// ----------------------------------------------------
// Calculate maximum expected current
// ----------------------------------------------------
IF in_lrHeaterResistance > 0.0 THEN
    stat.lrMaxCurrent := SQRT(in_lrHeaterMaxPower / in_lrHeaterResistance);
ELSE
    stat.lrMaxCurrent := 999.9;
END_IF;


// ----------------------------------------------------
// Calculate expected heater power and power ratio
// ----------------------------------------------------
lrExpectedPower :=
    (stat.lrActSetpoint / 100.0) * in_lrHeaterMaxPower;

stat.lrExpectedHeaterPower := lrExpectedPower;

IF lrExpectedPower > 0.0 THEN
    lrPowerRatio := stat.lrActHeaterPower / lrExpectedPower;
ELSE
    lrPowerRatio := 1.0;
END_IF;

stat.lrHeaterPowerRatio := lrPowerRatio;


// ----------------------------------------------------
// Heater open-loop detection
// ----------------------------------------------------
// Below 1% demand, current measurement is not reliable enough.
stat.bHeaterOpenLoop :=
    (lrPowerRatio < 0.10)
    AND stat.bActive
    AND stat.lrActSetpoint > 1.0;


// ----------------------------------------------------
// Heater short-circuit detection
// ----------------------------------------------------
stat.bHeaterShort :=
    stat.lrActCurrent > (stat.lrMaxCurrent + 1.0);


// ----------------------------------------------------
// Thermal switch open detection
// ----------------------------------------------------
// One or more parallel heater branches may be disconnected.
// Actual power is reduced, but not zero.
bThermalSwitchOpenCandidate :=
    (lrPowerRatio >= 0.10)
    AND (lrPowerRatio < 0.85)
    AND stat.bActive
    AND stat.lrActSetpoint > 10.0
    AND NOT stat.bHeaterOpenLoop
    AND NOT stat.bHeaterShort;

// Debounce to avoid false alarms during transients
tonThermalSwitchOpen(
    IN := bThermalSwitchOpenCandidate,
    PT := T#10s
);

stat.bHeaterThermalSwitchOpen := tonThermalSwitchOpen.Q;


// ----------------------------------------------------
// Insufficient heater power
// ----------------------------------------------------
// Heater demand is high, but delivered power is too low.
// This means the heater may not be able to reach/hold setpoint.
stat.bHeaterInsufficientPower :=
    stat.bActive
    AND stat.lrActSetpoint > 50.0
    AND (lrPowerRatio < 0.70)
    AND NOT stat.bHeaterOpenLoop
    AND NOT stat.bHeaterShort;


// ----------------------------------------------------
// General error / warning flags
// ----------------------------------------------------
stat.bError :=
    stat.bHwError
    OR stat.bHeaterOpenLoop
    OR stat.bHeaterShort
    OR stat.bHeaterThermalSwitchOpen
    OR stat.bHeaterInsufficientPower;

stat.bWarning := stat.bHwWarning;


// ----------------------------------------------------
// Store auto setpoint information
// ----------------------------------------------------
stat.lrAutoSetpointValue := in_lrAutoSetpointValue;
stat.sAutoSetpointSource := in_sAutoSetpointSource;


// ----------------------------------------------------
// Set heater state
// ----------------------------------------------------
IF stat.bHwError THEN
    stat.nHeaterState := E_METIS_CRYO_HEATER_STATE.ERROR;
    stat.sHeaterState := 'HW ERROR';

ELSIF stat.bHeaterShort THEN
    stat.nHeaterState := E_METIS_CRYO_HEATER_STATE.ERROR;
    stat.sHeaterState := 'HEATER SHORT CIRCUIT';

ELSIF stat.bHeaterOpenLoop THEN
    stat.nHeaterState := E_METIS_CRYO_HEATER_STATE.ERROR;
    stat.sHeaterState := 'HEATER OPEN CIRCUIT';

ELSIF stat.bHeaterThermalSwitchOpen THEN
    stat.nHeaterState := E_METIS_CRYO_HEATER_STATE.ERROR;
    stat.sHeaterState := 'THERMAL SWITCH OPEN';

ELSIF stat.bHeaterInsufficientPower THEN
    stat.nHeaterState := E_METIS_CRYO_HEATER_STATE.ERROR;
    stat.sHeaterState := 'INSUFFICIENT HEATER POWER';

ELSIF stat.bHwWarning THEN
    stat.nHeaterState := E_METIS_CRYO_HEATER_STATE.ERROR;
    stat.sHeaterState := 'HW WARNING';

ELSIF stat.bWarning THEN
    stat.nHeaterState := E_METIS_CRYO_HEATER_STATE.ERROR;
    stat.sHeaterState := 'WARNING';

ELSIF stat.bManual THEN
    stat.nHeaterState := E_METIS_CRYO_HEATER_STATE.ON;
    stat.sHeaterState := 'MANUAL';

ELSIF stat.bActive THEN
    stat.nHeaterState := E_METIS_CRYO_HEATER_STATE.ON;
    stat.sHeaterState := 'ON';

ELSE
    stat.nHeaterState := E_METIS_CRYO_HEATER_STATE.OFF;
    stat.sHeaterState := 'OFF';
END_IF;


M_SetStatus := NOT stat.bError;


// stat.lrAutoCtrlOut := in_lrAutoSetpointValue;
// 
// 
// CASE in_eHeaterType OF
//     
//     E_METIS_CRYO_HEATER_TYPE.PWM_DETECTOR,
//     E_METIS_CRYO_HEATER_TYPE.PWM_WINDOW:
//         // Set actual power I * 24.0V
//         stat.lrActHeaterPower := stat.lrActCurrent * stat.lrActCurrent * in_lrHeaterResistance;
// 
//     E_METIS_CRYO_HEATER_TYPE.PWM_SORPTION:
//     
//         // Set actual power I^(Average PWM Voltage)
//         // TODO : CHECK IF CORRECT
//         stat.lrActHeaterPower := ((stat.lrActCurrent * 24 * stat.lrActDutyCycle)/100);
// 
//     E_METIS_CRYO_HEATER_TYPE.CPAU60:
//         // Set actual power I^2R
//         stat.lrActHeaterPower := stat.lrActCurrent * stat.lrActCurrent * in_lrHeaterResistance;
//         
//     E_METIS_CRYO_HEATER_TYPE.CXWUI60:
//         // Set actual power I^2R
//         stat.lrActHeaterPower := stat.lrActCurrent * stat.lrActCurrent * in_lrHeaterResistance;
// 
//     E_METIS_CRYO_HEATER_TYPE.EL95X1:
//         IF stat.bActive THEN
//             stat.lrActHeaterPower := stat.lrActCurrent * stat.lrActVoltage;
//         ELSE
//             stat.lrActHeaterPower := 0.0;
//         END_IF
//         
// END_CASE
// 
// // Set max current
// IF in_lrHeaterResistance > 0.0 THEN
//     stat.lrMaxCurrent :=  SQRT(in_lrHeaterMaxPower/in_lrHeaterResistance);
// ELSE
//     stat.lrMaxCurrent := 999.9;
// END_IF
// 
// // check if the heater is in open loop
// // Note: below 1.00% the current measurement is not accurate, so don't report an open loop error!
// stat.bHeaterOpenLoop := (stat.lrActHeaterPower < 0.1 * (stat.lrActSetpoint/100.0) * in_lrHeaterMaxPower) // actual power in [W] is less than 10% of the expected power in [W]
//                         AND stat.bActive 
//                         AND stat.lrActSetpoint > 1.0; // lrActSetpoint is more than 1% 
// 
// // Check if there is a short circuit: Comparing the actual current with the Max current + 1 A  
// stat.bHeaterShort := stat.lrActCurrent > (stat.lrMaxCurrent + 1);
// 
// // calculate the general bError/bWarning flags
// stat.bError := stat.bHwError OR stat.bHeaterOpenLoop OR stat.bHeaterShort;
// stat.bWarning := stat.bHwWarning;
// 
// stat.lrAutoSetpointValue := in_lrAutoSetpointValue;
// stat.sAutoSetpointSource := in_sAutoSetpointSource;
// 
// IF stat.bHwError THEN
//     stat.nHeaterState := E_METIS_CRYO_HEATER_STATE.ERROR;
//     stat.sHeaterState := 'HW ERROR';
// ELSIF stat.bHwWarning THEN
//     stat.nHeaterState := E_METIS_CRYO_HEATER_STATE.ERROR;
//     stat.sHeaterState := 'HW WARNING';
// ELSIF stat.bHeaterOpenLoop THEN
//     stat.nHeaterState := E_METIS_CRYO_HEATER_STATE.ERROR;
//     stat.sHeaterState := 'HEATER OPEN LOOP ERROR';
// ELSIF stat.bHeaterShort THEN
//     stat.nHeaterState := E_METIS_CRYO_HEATER_STATE.ERROR;
//     stat.sHeaterState := 'HEATER SHORT ERROR';
// ELSIF stat.bError THEN
//     stat.nHeaterState := E_METIS_CRYO_HEATER_STATE.ERROR;
//     stat.sHeaterState := 'ERROR';
// ELSIF stat.bWarning THEN
//     stat.nHeaterState := E_METIS_CRYO_HEATER_STATE.ERROR;
//     stat.sHeaterState := 'WARNING';
// ELSIF stat.bActive THEN
//     stat.nHeaterState := E_METIS_CRYO_HEATER_STATE.ON;
//     stat.sHeaterState := 'ON';
// ELSE
//     stat.nHeaterState := E_METIS_CRYO_HEATER_STATE.OFF;
//     stat.sHeaterState := 'OFF';
// END_IF
// 
//
END_METHOD

METHOD M_UpdateAlarms
VAR_INPUT
END_VAR
VAR
	stEventEntry : TcEventEntry;
	sText : STRING;
END_VAR
//
// Set / clear alarms
//

fbAlarmHandler.M_UpdateAlarm(
    in_bCondition    := stat.bHeaterShort,
    in_nIndex        := 0,
    in_strEventEntry := Tc_Events.METISCryoHeaterEventClass.HeaterShortCircuit
);

fbAlarmHandler.M_UpdateAlarm(
    in_bCondition    := stat.bHeaterOpenLoop,
    in_nIndex        := 1,
    in_strEventEntry := Tc_Events.METISCryoHeaterEventClass.HeaterOpenCircuit
);

fbAlarmHandler.M_UpdateAlarm(
    in_bCondition    := stat.bManual,
    in_nIndex        := 2,
    in_strEventEntry := Tc_Events.METISCryoHeaterEventClass.HeaterManualMode
);

fbAlarmHandler.M_UpdateAlarm(
    in_bCondition    := stat.bHeaterThermalSwitchOpen,
    in_nIndex        := 3,
    in_strEventEntry := Tc_Events.METISCryoHeaterEventClass.HeaterThermalSwitchOpen
);

fbAlarmHandler.M_UpdateAlarm(
    in_bCondition    := stat.bHeaterInsufficientPower,
    in_nIndex        := 4,
    in_strEventEntry := Tc_Events.METISCryoHeaterEventClass.HeaterInsufficientPower
);


//
// Handle alarms
//
fbAlarmHandler(stAlarms := stat.stAlarms);

fbAlarmHandler.M_ProcessAlarms(
    arrEventEntry := arrEventEntry,
    sEventString  := in_sName
);

// //
// // Set / clear alarms
// //
// 
// // Global alarm if the voted temperature reading is not valid.
// fbAlarmHandler.M_UpdateAlarm(
//     in_bCondition    := stat.bHeaterOpenLoop,
//     in_nIndex        := 1,
//     in_strEventEntry := Tc_Events.METISCryoHeaterEventClass.HeaterOpenCircuit
// );
// 
// 
// fbAlarmHandler.M_UpdateAlarm(
//     in_bCondition    := stat.bHeaterShort,
//     in_nIndex        := 0,
//     in_strEventEntry := Tc_Events.METISCryoHeaterEventClass.HeaterShortCircuit
// );
// 
// fbAlarmHandler.M_UpdateAlarm(
//     in_bCondition    := stat.bManual,
//     in_nIndex        := 2,
//     in_strEventEntry := Tc_Events.METISCryoHeaterEventClass.HeaterManualMode
// );
// 
// fbAlarmHandler.M_UpdateAlarm(
//     in_bCondition    := stat.,
//     in_nIndex        := 3,
//     in_strEventEntry := Tc_Events.METISCryoHeaterEventClass.HeaterThermalSwitchOpen
// );
// 
// fbAlarmHandler.M_UpdateAlarm(
//     in_bCondition    := stat.,
//     in_nIndex        := 4,
//     in_strEventEntry := Tc_Events.METISCryoHeaterEventClass.HeaterInsufficientPower
// );
// 
// 
// 
// 
// 
// //
// // Handle alarms
// //
// fbAlarmHandler(stAlarms := stat.stAlarms);
// 
// fbAlarmHandler.M_ProcessAlarms(
//     arrEventEntry := arrEventEntry,
//     sEventString  := in_sName
// );
END_METHOD

END_FUNCTION_BLOCK

// POUs/XML_Cfg_Read_Write/FB_READ_WRITE_HEATER_CONFIG
FUNCTION_BLOCK FB_READ_WRITE_HEATER_CONFIG EXTENDS FB_READ_WRITE_CONFIG_BASE
VAR_INPUT
	in_sHeaterName:      T_MaxString;
END_VAR
VAR_IN_OUT
	cfg:   T_METIS_HEATER_CFG;
END_VAR

SUPER^(
    in_sEntryName  := in_sHeaterName,
    in_sSubFolder  := 'Heater\',
    in_sXPath      := '/Heater_Configuration/',
    in_pSymAddr    := ADR(cfg),
    in_cbSymSize   := SIZEOF(cfg));

END_FUNCTION_BLOCK

// POUs/Devices/Control_Valves_Ctrl/FB_METIS_CONTROL_VALVE
FUNCTION_BLOCK FB_METIS_CONTROL_VALVE
VAR_INPUT
    {attribute 'OPC.UA.DA' := '0'}    
    in_sName:               STRING  := 'Ctrl Valve'; // Valve name
//    {attribute 'OPC.UA.DA' := '0'}
//    in_lrHeaterResistance:  LREAL;               // Resistance of the heater to be controlled [Ohms]
//    {attribute 'OPC.UA.DA' := '0'}
//    in_lrHeaterMaxPower:    LREAL;               // Max power of the heater to be controlled [Watts]    
    {attribute 'OPC.UA.DA' := '0'}

    in_eValveType:         		E_METIS_CRYO_CTRL_VALVE_TYPE := E_METIS_CRYO_Ctrl_VALVE_TYPE.NONE;
    {attribute 'OPC.UA.DA' := '0'}

    in_sAutoSetpointSource:     STRING;          // Name of the source of the AUTO setpoint
    
    {attribute 'OPC.UA.DA' := '0'}
    in_bEnable : BOOL;                           // Auto-mode enable
    
   {attribute 'OPC.UA.DA' := '0'}
   in_lrAutoSetpointValue:     LREAL;           // Output power coming for the AUTO setpoint
END_VAR
VAR
(*TODO: This input is useful if a PID ctrl loop is implemeted to control the valve.
For the moment, There are three set points, Off, Normal and Alarm*)	
// 	{attribute 'OPC.UA.DA' := '0'}
//     in_lrAutoSetpointValue:     LREAL;           // Output power coming for the AUTO setpoint
    {attribute 'OPC.UA.DA' := '0'}
    nTimeout:                   UDINT := 10000;     // Timeout for current to change [ms] after enabling power. Default 10000.
    {attribute 'OPC.UA.DA' := '0'}
	{attribute 'TcHmiSymbol.Show'}
    bInterlock:                 BOOL := FALSE;      // External Interlock
    {attribute 'OPC.UA.DA' := '0'}
    i_nCouplerState     AT %I*: UINT;               // Terminal state. Should be 8, i.e. OP.
// Hardware link    
    {attribute 'OPC.UA.DA' := '0'}
    io_anti_fog_blower      : T_METIS_CTRL_VALVE_IO_ANTI_FOG_BLOWER;
    {attribute 'OPC.UA.DA' := '0'}
    io_img_cfo_precooling   : T_METIS_CTRL_VALVE_IO_IMG_CFO_PRECOOLING;
    // EL2819 diagnostics for the output channel

    i_bOverTemperature  AT %I*: BOOL;
    i_bOpenLoad         AT %I*: BOOL;
    i_bOverCurrent      AT %I*: BOOL;
    i_bShortTo24V       AT %I*: BOOL;
	
//    {attribute 'OPC.UA.DA' := '0'}
//    io_cxwui60  : T_METIS_HEATER_IO_CXWUI60;
    
    {attribute 'OPC.UA.DA' := '1'}
	{attribute 'TcHmiSymbol.Show'}
    stat:        T_METIS_CTRL_VALVE_STAT;
    {attribute 'OPC.UA.DA' := '1'}
	{attribute 'TcHmiSymbol.ShowRecursively'}
    ctrl:        T_METIS_CTRL_VALVE_CTRL;
    {attribute 'OPC.UA.DA' := '1'}
	{attribute 'TcHmiSymbol.Show'}
		{attribute 'TcHmiSymbol.ShowRecursively'}
    cfg:         T_METIS_CTRL_VALVE_CFG;

    {attribute 'OPC.UA.DA' := '0'}
	{attribute 'TcHmiSymbol.Show'}
    fbConfig    : FB_READ_WRITE_CONTROL_VALVE_CONFIG; 
	
				// Alarm handling
	// List of alarms to be handled by Temperature
	arrEventEntry : ARRAY [0..3] OF TcEventEntry;
	// Alarm handler FB
	fbAlarmHandler : FB_AlarmHandler;
	{attribute 'TcHmiSymbol.Show'}
	{attribute 'TcHmiSymbol.ReadOnly'}
	sInstanceName : T_MaxString;
	{attribute 'TcHmiSymbol.Show'}
	bConfirmAllAlarms : BOOL;
	{attribute 'TcHmiSymbol.Show'}
	{attribute 'TcHmiSymbol.ReadOnly'}
	sEventClassName : T_MaxString;
	
	// Logs logs
	logs:	FB_CRYO_FUNCTION_LOG;
    
END_VAR

IF not stat.bConfigured THEN
    M_Configure();
END_IF

// Read/write the configuration
fbConfig(in_sCtrlValveName:= in_sName, cfg := cfg);

M_SetMode();

M_UpdateActive();

M_ReadInputs();

M_SetStatus();

M_SetCtrlOutput();

// read/write the config (if needed)
M_Read_Write_Config();

// Handle alarms
M_UpdateAlarms();

METHOD M_Activity_Valve_Alarm : BOOL
VAR_INPUT
END_VAR
in_lrAutoSetpointValue := cfg.lrBlowerAlarmSetPoint;
END_METHOD

METHOD M_Activity_Valve_None : BOOL
VAR_INPUT
END_VAR
in_lrAutoSetpointValue := 0.0;
END_METHOD

METHOD M_Activity_Valve_Normal : BOOL
VAR_INPUT
END_VAR
in_lrAutoSetpointValue := cfg.lrBlowerNormalSetPoint;
END_METHOD

METHOD M_Configure
VAR_INPUT
END_VAR
VAR_INST
    {attribute 'OPC.UA.DA' := '0'}
    nConfigureState : INT;
END_VAR
arrEventEntry[0] := Tc_Events.METISCryoCtrlValveEventClass.ValveOpenLoad;
arrEventEntry[1] := Tc_Events.METISCryoCtrlValveEventClass.ValveShortCircuit;
arrEventEntry[2] := Tc_Events.METISCryoCtrlValveEventClass.ValveManualMode;
arrEventEntry[3] := Tc_Events.METISCryoCtrlValveEventClass.ValveFeedbackFailure;


CASE nConfigureState OF
    0:  
        // set some defaults
        stat.eCtrlMode := E_METIS_CTRL_MODE.AUTO;   // always start in AUTO mode
        cfg.lrAutoScalePercent := 100.0;            // 100% by default
        
        // start reading the config
        fbConfig.M_ReadConfiguration();
        nConfigureState := 1;
    1:
        IF fbConfig.bReadingDoneFlag THEN
            
            // clear the flag
            fbConfig.M_ClearReadingDoneFlag();
            
            // set the bConfigured flag
            stat.bConfigured := TRUE;

        END_IF
END_CASE
END_METHOD

METHOD M_GetError : BOOL
VAR_INPUT
    m_nAI_HWStatus : UINT;
END_VAR
VAR_INST
    tonErrorEnableDelay : TON;
    tErrorEnableDelay   : TIME := T#5S;
END_VAR
VAR
    bUseAnalogFeedback : BOOL;
END_VAR
M_GetError := FALSE;


// ----------------------------------------------------
// Reset accepted error flags every cycle
// ----------------------------------------------------
stat.bValveOpenLoadError     := FALSE;
stat.bValveShortCircuitError := FALSE;
stat.bValveFeedbackError     := FALSE;


// ----------------------------------------------------
// Valve-type dependent feedback
// ----------------------------------------------------
CASE in_eValveType OF

    E_METIS_CRYO_CTRL_VALVE_TYPE.ANTI_FOG_BLOWER:
        bUseAnalogFeedback := TRUE;

    E_METIS_CRYO_CTRL_VALVE_TYPE.PRE_COOLING_IMG_CFO:
        bUseAnalogFeedback := FALSE;

ELSE
    bUseAnalogFeedback := FALSE;

END_CASE;


// ----------------------------------------------------
// Always read EL2819 diagnostics for both valve types
// ----------------------------------------------------
stat.bOpenLoad        := i_bOpenLoad;
stat.bShortTo24V      := i_bShortTo24V;
stat.bOverCurrent     := i_bOverCurrent;
stat.bOverTemperature := i_bOverTemperature;


// ----------------------------------------------------
// Read EL3124 analog feedback diagnostics only
// for valves that actually have analog feedback
// ----------------------------------------------------
IF bUseAnalogFeedback THEN
    stat.bInputUnder := (m_nAI_HWStatus AND 2#0000_0000_0000_0001) <> 0;
    stat.bInputOver  := (m_nAI_HWStatus AND 2#0000_0000_0000_0010) <> 0;
    stat.bHWError    := (m_nAI_HWStatus AND 2#0000_0000_0100_0000) <> 0;
ELSE
    stat.bInputUnder := FALSE;
    stat.bInputOver  := FALSE;
    stat.bHWError    := FALSE;
END_IF;


// ----------------------------------------------------
// Error evaluation only when valve is enabled,
// after startup delay
// ----------------------------------------------------
IF in_bEnable THEN

    tonErrorEnableDelay(IN := TRUE, PT := tErrorEnableDelay);

    IF tonErrorEnableDelay.Q THEN

        IF stat.bOpenLoad THEN
            stat.bError := TRUE;
            stat.bValveOpenLoadError := TRUE;
            stat.sValveState := 'OPEN LOAD';

        ELSIF stat.bShortTo24V OR stat.bOverCurrent OR stat.bOverTemperature THEN
            stat.bError := TRUE;
            stat.bValveShortCircuitError := TRUE;

            IF stat.bShortTo24V THEN
                stat.sValveState := 'SHORT TO 24V';
            ELSIF stat.bOverCurrent THEN
                stat.sValveState := 'OVERCURRENT';
            ELSE
                stat.sValveState := 'OVERTEMPERATURE';
            END_IF

        ELSIF bUseAnalogFeedback AND (stat.bHWError OR stat.bInputUnder OR stat.bInputOver) THEN
            stat.bError := TRUE;
            stat.bValveFeedbackError := TRUE;

            IF stat.bHWError THEN
                stat.sValveState := 'AI HW ERROR';
            ELSIF stat.bInputUnder THEN
                stat.sValveState := 'AI INPUT UNDERRANGE';
            ELSE
                stat.sValveState := 'AI INPUT OVERRANGE';
            END_IF

        ELSE
            stat.bError := FALSE;
        END_IF

    ELSE
        // Valve just enabled; ignore temporary diagnostics
        stat.bError := FALSE;
    END_IF

ELSE
    // Valve disabled; expected diagnostics are ignored
    tonErrorEnableDelay(IN := FALSE);
    stat.bError := FALSE;
END_IF


M_GetError := stat.bError;
END_METHOD

METHOD M_IsValveInError : BOOL
VAR_INPUT
END_VAR
M_IsValveInError := stat.bError;
END_METHOD

METHOD M_Read_Write_Config
VAR_INPUT
END_VAR
VAR_IN_OUT
END_VAR

IF ctrl.bWriteConfig THEN
    
    // (update the cfg object if needed)
    // ...
    
    // write the cfg object
    fbConfig.M_WriteConfiguration();
    ctrl.bWriteConfig := FALSE;
            
ELSIF ctrl.bReadConfig THEN

    fbConfig.M_ReadConfiguration();
    ctrl.bReadConfig := FALSE;
    
END_IF


IF fbConfig.bReadingDoneFlag THEN
    // clear the flag
    fbConfig.M_ClearReadingDoneFlag();
END_IF
END_METHOD

METHOD M_ReadInputs
VAR_INPUT
END_VAR
VAR
END_VAR
(*
    Read all inputs and assign values to variables.
*)

CASE in_eValveType OF
    
    E_METIS_CRYO_CTRL_VALVE_TYPE.ANTI_FOG_BLOWER:
	
        M_ScaleInput(m_nActCurrent:= io_anti_fog_blower.i_nFlowFeedBackCurrent);
        M_GetError(m_nAI_HWStatus := io_anti_fog_blower.i_nFeedBackStatus);
                

    E_METIS_CRYO_CTRL_VALVE_TYPE.PRE_COOLING_IMG_CFO:
        ;

   

END_CASE
END_METHOD

METHOD M_ScaleInput : BOOL
VAR_INPUT
    m_nActCurrent:    DINT;
END_VAR
VAR
    nActCurrentClamped : DINT;
    lrCtrlFlowClamped  : LREAL;
END_VAR
M_ScaleInput := FALSE;

// Clamp requested value
lrCtrlFlowClamped := stat.lrActSetpoint;

IF lrCtrlFlowClamped < 0.0 THEN
    lrCtrlFlowClamped := 0.0;
ELSIF lrCtrlFlowClamped > 100.0 THEN
    lrCtrlFlowClamped := 100.0;
END_IF


CASE in_eValveType OF

    E_METIS_CRYO_CTRL_VALVE_TYPE.ANTI_FOG_BLOWER:

        // Clamp raw feedback input
        nActCurrentClamped := m_nActCurrent;

        IF nActCurrentClamped < 0 THEN
            nActCurrentClamped := 0;
        ELSIF nActCurrentClamped > 32767 THEN
            nActCurrentClamped := 32767;
        END_IF

        // Convert real 4...20 mA feedback to valve opening [%]
        stat.lrActValveFlow :=
            DINT_TO_LREAL(nActCurrentClamped) * 100.0 / 32767.0;

        M_ScaleInput := TRUE;


    E_METIS_CRYO_CTRL_VALVE_TYPE.PRE_COOLING_IMG_CFO:

        // No active feedback available.
        // HMI displays requested value as assumed actual valve position.
        stat.lrActValveFlow := lrCtrlFlowClamped;

        M_ScaleInput := TRUE;


ELSE
    stat.lrActValveFlow := 0.0;
    M_ScaleInput := FALSE;

END_CASE
END_METHOD

METHOD M_ScaleOutput : BOOL
VAR_INPUT
    lrCtrlFlow : LREAL; // Requested valve opening [%], 0.0 ... 100.0
END_VAR
VAR
    lrCtrlFlowClamped : LREAL;
    nOutputRaw        : INT;
END_VAR

M_ScaleOutput := FALSE;

// Clamp command to valid range
lrCtrlFlowClamped := lrCtrlFlow;

IF lrCtrlFlowClamped < 0.0 THEN
    lrCtrlFlowClamped := 0.0;
ELSIF lrCtrlFlowClamped > 100.0 THEN
    lrCtrlFlowClamped := 100.0;
END_IF

// EL4124: 4...20 mA range.
// Assumption: 0 raw = 4 mA, 32767 raw = 20 mA.
nOutputRaw := LREAL_TO_INT(lrCtrlFlowClamped * 32767.0 / 100.0);

CASE in_eValveType OF

    E_METIS_CRYO_CTRL_VALVE_TYPE.ANTI_FOG_BLOWER:
        io_anti_fog_blower.q_nSetCurrent := nOutputRaw;
        M_ScaleOutput := TRUE;

    E_METIS_CRYO_CTRL_VALVE_TYPE.PRE_COOLING_IMG_CFO:
        io_img_cfo_precooling.q_nSetCurrent := nOutputRaw;
        M_ScaleOutput := TRUE;

ELSE
    M_ScaleOutput := FALSE;
END_CASE
END_METHOD

METHOD M_SetCtrlOutput : BOOL
VAR 
END_VAR
CASE in_eValveType OF
    
    E_METIS_CRYO_CTRL_VALVE_TYPE.ANTI_FOG_BLOWER:

		M_ScaleOutput(lrCtrlFlow := stat.lrActSetpoint);
        
    E_METIS_CRYO_CTRL_VALVE_TYPE.PRE_COOLING_IMG_CFO:
			M_ScaleOutput(lrCtrlFlow := stat.lrActSetpoint);
    




END_CASE
END_METHOD

// Disable the controller in auto mode
METHOD M_SetDisable
VAR_INPUT
END_VAR
in_bEnable := FALSE;

M_UpdateActive();
END_METHOD

// Enable the controller in auto mode
METHOD M_SetEnable
VAR_INPUT
END_VAR
in_bEnable := TRUE;

M_UpdateActive();
END_METHOD

METHOD M_SetManualDisable
ctrl.bManualEnable := FALSE;

M_UpdateActive();
END_METHOD

METHOD M_SetManualEnable : BOOL
ctrl.bManualEnable := TRUE;

M_UpdateActive();
END_METHOD

METHOD M_SetMode
VAR_INPUT
END_VAR
If stat.eCtrlMode = E_METIS_CTRL_MODE.NONE THEN
    // typical behavior when e.g. a config file did not contain a valid entry
    // To avoid problems, force MANUAL in this case
    stat.eCtrlMode := E_METIS_CTRL_MODE.MANUAL;
END_IF

// check which mode switches are accepted
// (currently very simple, but can be made more complex if needed)
stat.bAcceptCtrlMode_Auto := stat.eCtrlMode = E_METIS_CTRL_MODE.MANUAL
                             AND NOT stat.bError;
stat.bAcceptCtrlMode_Manual := stat.eCtrlMode = E_METIS_CTRL_MODE.AUTO ;

// switch to AUTO / MANUAL mode if acceptable
IF ctrl.eCtrlMode = E_METIS_CTRL_MODE.AUTO AND stat.bAcceptCtrlMode_Auto THEN
    stat.eCtrlMode := E_METIS_CTRL_MODE.AUTO;
ELSIF ctrl.eCtrlMode = E_METIS_CTRL_MODE.MANUAL AND stat.bAcceptCtrlMode_Manual THEN
    stat.eCtrlMode := E_METIS_CTRL_MODE.MANUAL;
END_IF

// update the redundant booleans (for easy HMI development)
stat.bAuto   := stat.eCtrlMode = E_METIS_CTRL_MODE.AUTO;
stat.bManual := stat.eCtrlMode = E_METIS_CTRL_MODE.MANUAL;

// update the actual setpoint
IF stat.bAuto THEN
    stat.lrActSetpoint := (in_lrAutoSetpointValue * LIMIT(0, cfg.lrAutoScalePercent, 100))/100; // dividing by 100 to debug % setpoint error
ELSIF stat.bManual THEN
    stat.lrActSetpoint := ctrl.lrManualSetpoint;
ELSE
    stat.lrActSetpoint := 0.0;
END_IF

// reset any request
ctrl.eCtrlMode := E_METIS_CTRL_MODE.NONE;
END_METHOD

METHOD M_SetStatus : BOOL
VAR_INPUT
END_VAR
M_SetStatus := FALSE;

stat.sName := in_sName;

stat.lrAutoCtrlOut := in_lrAutoSetpointValue;
stat.lrAutoSetpointValue := in_lrAutoSetpointValue;
stat.sAutoSetpointSource := in_sAutoSetpointSource;

sInstanceName := fbAlarmHandler.sInstanceName;
sEventClassName := fbAlarmHandler.sEventClassName;
IF bConfirmAllAlarms THEN
	bConfirmAllAlarms := FALSE;
	fbAlarmHandler.M_ConfirmAllAlarms();
END_IF



CASE in_eValveType OF

    E_METIS_CRYO_CTRL_VALVE_TYPE.ANTI_FOG_BLOWER:
        ;

    E_METIS_CRYO_CTRL_VALVE_TYPE.PRE_COOLING_IMG_CFO:
        ;

END_CASE

IF stat.bError THEN
    stat.nValveState := E_METIS_CRYO_CTRL_VALVE_STATE.ERROR;

//     // Keep detailed message from M_GetError 
//     IF stat.sValveState = '' THEN
//         stat.sValveState := 'ERROR';
//     END_IF

ELSIF stat.bWarning THEN
    stat.nValveState := E_METIS_CRYO_CTRL_VALVE_STATE.ERROR;
    stat.sValveState := 'WARNING';

ELSIF stat.bActive THEN
    stat.nValveState := E_METIS_CRYO_CTRL_VALVE_STATE.ON;
    stat.sValveState := 'ON';

ELSE
    stat.nValveState := E_METIS_CRYO_CTRL_VALVE_STATE.OFF;
    stat.sValveState := 'OFF';
END_IF

M_SetStatus := NOT stat.bError;
END_METHOD

METHOD M_UpdateActive
VAR_INPUT
END_VAR

IF stat.bAuto THEN
    stat.bActive := in_bEnable;
ELSIF stat.bManual THEN
    stat.bActive := ctrl.bManualEnable;
END_IF

CASE in_eValveType OF
 
    E_METIS_CRYO_CTRL_VALVE_TYPE.ANTI_FOG_BLOWER:
	
        io_anti_fog_blower.q_bEnable := stat.bActive;
// 		io_anti_fog_purge.q_bEnable := stat.bActive;
    
	E_METIS_CRYO_CTRL_VALVE_TYPE.PRE_COOLING_IMG_CFO:
	;
	 
END_CASE
END_METHOD

METHOD M_UpdateAlarms
VAR_INPUT
END_VAR
VAR
	stEventEntry : TcEventEntry;
	sText : STRING;
END_VAR
//
// Set / clear alarms
//

fbAlarmHandler.M_UpdateAlarm(
    in_bCondition    := stat.bValveOpenLoadError,
    in_nIndex        := 0,
    in_strEventEntry := Tc_Events.METISCryoCtrlValveEventClass.ValveOpenLoad
);

fbAlarmHandler.M_UpdateAlarm(
    in_bCondition    := stat.bValveShortCircuitError,
    in_nIndex        := 1,
    in_strEventEntry := Tc_Events.METISCryoCtrlValveEventClass.ValveShortCircuit
);

fbAlarmHandler.M_UpdateAlarm(
    in_bCondition    := stat.bManual,
    in_nIndex        := 2,
    in_strEventEntry := Tc_Events.METISCryoCtrlValveEventClass.ValveManualMode
);

fbAlarmHandler.M_UpdateAlarm(
    in_bCondition    := stat.bValveFeedbackError,
    in_nIndex        := 3,
    in_strEventEntry := Tc_Events.METISCryoCtrlValveEventClass.ValveFeedbackFailure
);


//
// Handle alarms
//
fbAlarmHandler(stAlarms := stat.stAlarms);

fbAlarmHandler.M_ProcessAlarms(
    arrEventEntry := arrEventEntry,
    sEventString  := in_sName
);
END_METHOD

END_FUNCTION_BLOCK

// POUs/XML_Cfg_Read_Write/FB_READ_WRITE_CONTROL_VALVE_CONFIG
FUNCTION_BLOCK FB_READ_WRITE_CONTROL_VALVE_CONFIG EXTENDS FB_READ_WRITE_CONFIG_BASE
VAR_INPUT
	in_sCtrlValveName:      T_MaxString;
END_VAR
VAR_IN_OUT
	cfg:   T_METIS_CTRL_VALVE_CFG;
END_VAR

SUPER^(
    in_sEntryName  := in_sCtrlValveName,
    in_sSubFolder  := 'Control_Valve\',
    in_sXPath      := '/CtrlValve_Configuration/',
    in_pSymAddr    := ADR(cfg),
    in_cbSymSize   := SIZEOF(cfg));

END_FUNCTION_BLOCK

// HMI/POUs/Cryo-Routines/Cool-Down/FB_HMI_COOL_DOWN
FUNCTION_BLOCK FB_HMI_COOL_DOWN EXTENDS FB_HMI_COMPONENT
VAR_INPUT
END_VAR
VAR_OUTPUT
END_VAR
VAR
END_VAR
VAR_IN_OUT
	{attribute 'OPC.UA.DA' := '0'}
	fbInstance		: FB_METIS_CRYO_COOL_DOWN;
	{attribute 'OPC.UA.DA' := '0'}
	interlocks:						T_METIS_CRYO_INTERLOCKS;

END_VAR


fbHealthStatus( 
				bIsEnabled:= TRUE, 
				bIsGood := NOT fbInstance.stat.bError,
				bHasWarning := fbInstance.stat.bWarning OR interlocks.bInterlock_CoolDown
				);
				
fbBusyStatus(
				bIsBusy := fbInstance.stat.bBusy,
				bIsEnabled := TRUE);
				
M_UpdateStatusColor();

END_FUNCTION_BLOCK

// HMI/POUs/Cryo-Routines/Evacuation/FB_HMI_EVACUATION
FUNCTION_BLOCK FB_HMI_EVACUATION EXTENDS FB_HMI_COMPONENT
VAR_INPUT
END_VAR
VAR_OUTPUT
END_VAR
VAR
END_VAR
VAR_IN_OUT
	{attribute 'OPC.UA.DA' := '0'}
	fbInstance		: FB_METIS_CRYO_EVAC;
	{attribute 'OPC.UA.DA' := '0'}
	interlocks:						T_METIS_CRYO_INTERLOCKS;

END_VAR


fbHealthStatus( 
				bIsEnabled:= TRUE, 
				bIsGood := NOT fbInstance.stat.bError,
				bHasWarning := fbInstance.stat.bWarning OR interlocks.bInterlock_Evacuation
				);
				
fbBusyStatus(
				bIsBusy := fbInstance.stat.bBusy,
				bIsEnabled := TRUE);
				
M_UpdateStatusColor();

END_FUNCTION_BLOCK

// HMI/POUs/Cryo-Routines/Power-Outage/FB_HMI_POWER_OUTAGE
FUNCTION_BLOCK FB_HMI_POWER_OUTAGE EXTENDS FB_HMI_COMPONENT
VAR_INPUT
END_VAR
VAR_OUTPUT
END_VAR
VAR
END_VAR

END_FUNCTION_BLOCK

// HMI/POUs/Cryo-Routines/Regeneration/FB_HMI_REGENERATION
FUNCTION_BLOCK FB_HMI_REGENERATION EXTENDS FB_HMI_COMPONENT
VAR_INPUT
END_VAR
VAR_OUTPUT
END_VAR
VAR
END_VAR
VAR_IN_OUT
	{attribute 'OPC.UA.DA' := '0'}
	fbInstance		: FB_METIS_CRYO_REGENERATION;
	{attribute 'OPC.UA.DA' := '0'}
	interlocks:						T_METIS_CRYO_INTERLOCKS;

END_VAR


fbHealthStatus( 
				bIsEnabled:= TRUE, 
				bIsGood := NOT fbInstance.stat.bError,
				bHasWarning := fbInstance.stat.bWarning OR interlocks.bInterlock_Regeneration
				);
				
fbBusyStatus(
				bIsBusy := fbInstance.stat.bBusy,
				bIsEnabled := TRUE);
				
M_UpdateStatusColor();

END_FUNCTION_BLOCK

// HMI/POUs/Cryo-Routines/Venting/FB_HMI_VENTING
FUNCTION_BLOCK FB_HMI_VENTING EXTENDS FB_HMI_COMPONENT
VAR_INPUT
END_VAR
VAR_OUTPUT
END_VAR
VAR
END_VAR
VAR_IN_OUT
	{attribute 'OPC.UA.DA' := '0'}
	fbInstance		: FB_METIS_CRYO_VENTING;
	{attribute 'OPC.UA.DA' := '0'}
	interlocks:						T_METIS_CRYO_INTERLOCKS;

END_VAR


fbHealthStatus( 
				bIsEnabled:= TRUE, 
				bIsGood := NOT fbInstance.stat.bError,
				bHasWarning := fbInstance.stat.bWarning OR interlocks.bInterlock_Venting
				);
				
fbBusyStatus(
				bIsBusy := fbInstance.stat.bBusy,
				bIsEnabled := TRUE);
				
M_UpdateStatusColor();

END_FUNCTION_BLOCK

// HMI/POUs/Cryo-Routines/Warm-Up/FB_HMI_WARM_UP
FUNCTION_BLOCK FB_HMI_WARM_UP EXTENDS FB_HMI_COMPONENT
VAR_INPUT
END_VAR
VAR_OUTPUT
END_VAR
VAR
END_VAR
VAR_IN_OUT
	{attribute 'OPC.UA.DA' := '0'}
	fbInstance		: FB_METIS_CRYO_WARM_UP;
	{attribute 'OPC.UA.DA' := '0'}
	interlocks:						T_METIS_CRYO_INTERLOCKS;

END_VAR


fbHealthStatus( 
				bIsEnabled:= TRUE, 
				bIsGood := NOT fbInstance.stat.bError,
				bHasWarning := fbInstance.stat.bWarning OR interlocks.bInterlock_WarmUp
				);
				
fbBusyStatus(
				bIsBusy := fbInstance.stat.bBusy,
				bIsEnabled := TRUE);
				
M_UpdateStatusColor();

END_FUNCTION_BLOCK

// HMI/POUs/Devices/Cabinets/FB_HMI_CABINETS
FUNCTION_BLOCK FB_HMI_CABINETS EXTENDS FB_HMI_COMPONENT
VAR_INPUT
END_VAR
VAR_OUTPUT
END_VAR
VAR
END_VAR

END_FUNCTION_BLOCK

// HMI/POUs/Devices/Cabinets/FB_HMI_CCU
FUNCTION_BLOCK FB_HMI_CCU EXTENDS FB_HMI_COMPONENT
VAR_INPUT
END_VAR
VAR_OUTPUT
END_VAR
VAR_IN_OUT
    fbInstance : FB_MET_CCU;
END_VAR
VAR
END_VAR

fbHealthStatus(
    bIsEnabled := TRUE,
    bIsGood :=      (NOT fbInstance.cooling.stat.bError)
                AND (NOT fbInstance.cooling.stat.bThermoswitchOpen)
                AND (NOT fbInstance.cooling.stat.bAlarm_Cabinet)
                AND (NOT fbInstance.cooling.stat.bFrontDoorOpen)
                AND (NOT fbInstance.cooling.stat.bRearDoorOpen)
                AND (NOT fbInstance.power.stat.bError)
                AND (fbInstance.power.stat.bNormalPower_ConditionsOK)
                AND (fbInstance.fuseSS.stat.nSubstate = E_FUSE_SUBSTATE.OP_ON)
                AND (fbInstance.fuseAux24V.stat.nSubstate = E_FUSE_SUBSTATE.OP_ON));

fbBusyStatus(
    bIsEnabled := FALSE,
    bIsBusy := FALSE);

M_UpdateStatusColor();

END_FUNCTION_BLOCK

// HMI/POUs/Devices/Control_Loops/FB_HMI_CONTROL_LOOPS
FUNCTION_BLOCK FB_HMI_CONTROL_LOOPS EXTENDS FB_HMI_COMPONENT
VAR_INPUT
END_VAR
VAR_OUTPUT
END_VAR
VAR
END_VAR

END_FUNCTION_BLOCK

// HMI/POUs/Devices/Control_Loops/FB_HMI_METIS_CTRL_TEMPERATURE
FUNCTION_BLOCK FB_HMI_METIS_CTRL_TEMPERATURE EXTENDS FB_HMI_COMPONENT
VAR_INPUT
END_VAR
VAR_OUTPUT
END_VAR
VAR_IN_OUT
    fbInstance : FB_METIS_CTRL_TEMPERATURE;
END_VAR
VAR
END_VAR

fbHealthStatus(
    bIsEnabled := fbInstance.cfg.bEnabled,
    bIsGood := fbInstance.stat.bValid);
                     
fbBusyStatus(
    bIsEnabled := FALSE,
    bIsBusy := FALSE);

M_UpdateStatusColor();

END_FUNCTION_BLOCK

// HMI/POUs/Devices/Control_Units/FB_HMI_CONTROL_UNITS
FUNCTION_BLOCK FB_HMI_CONTROL_UNITS EXTENDS FB_HMI_COMPONENT
VAR_INPUT
END_VAR
VAR_OUTPUT
END_VAR
VAR
END_VAR

END_FUNCTION_BLOCK

// HMI/POUs/Devices/Coolers/FB_HMI_COOLERS
FUNCTION_BLOCK FB_HMI_COOLERS EXTENDS FB_HMI_COMPONENT
VAR_INPUT
END_VAR
VAR_OUTPUT
END_VAR
VAR
END_VAR

END_FUNCTION_BLOCK

// HMI/POUs/Devices/Detectors/FB_HMI_DETECTORS
FUNCTION_BLOCK FB_HMI_DETECTORS EXTENDS FB_HMI_COMPONENT
VAR_INPUT
END_VAR
VAR_OUTPUT
END_VAR
VAR
END_VAR

END_FUNCTION_BLOCK

// HMI/POUs/Devices/Heaters/FB_HMI_HEATERS
FUNCTION_BLOCK FB_HMI_HEATERS EXTENDS FB_HMI_COMPONENT
VAR_INPUT
END_VAR
VAR_OUTPUT
END_VAR
VAR
END_VAR

END_FUNCTION_BLOCK

// HMI/POUs/Devices/Heaters/FB_HMI_METIS_HEATER
FUNCTION_BLOCK FB_HMI_METIS_HEATER EXTENDS FB_HMI_COMPONENT
VAR_INPUT
END_VAR
VAR_OUTPUT
END_VAR
VAR_IN_OUT
    fbInstance : FB_METIS_HEATER;
END_VAR
VAR
END_VAR

fbHealthStatus(
    bIsEnabled := fbInstance.stat.bActive,
    bIsGood := NOT fbInstance.stat.bError,
    bHasWarning := fbInstance.stat.bWarning);
                     
fbBusyStatus(
    bIsEnabled := FALSE,
    bIsBusy := FALSE);

M_UpdateStatusColor();

END_FUNCTION_BLOCK

// HMI/POUs/Devices/Lakeshores/FB_HMI_LAKESHORE
FUNCTION_BLOCK FB_HMI_LAKESHORE EXTENDS FB_HMI_COMPONENT
VAR_INPUT
    bConnected : BOOL;
END_VAR
VAR_OUTPUT
END_VAR
VAR_IN_OUT
    fbInstance : FB_METIS_LAKESHORE_336_TCP;
END_VAR
VAR
END_VAR

fbHealthStatus(
    bIsEnabled := bConnected,
    bIsGood := fbInstance.stat.nSubstate = E_RS_BASE_SUBSTATE.OP_MONITORING,
    bHasWarning := fbInstance.stat.bLocal);
                     
fbBusyStatus(
    bIsEnabled := bConnected,
    bIsBusy := fbInstance.stat.nSubstate = E_RS_BASE_SUBSTATE.NOTOP_INITIALIZING);

M_UpdateStatusColor();

END_FUNCTION_BLOCK

// HMI/POUs/Devices/Pressures/FB_HMI_PRESSURES
FUNCTION_BLOCK FB_HMI_PRESSURES EXTENDS FB_HMI_COMPONENT
VAR_INPUT
END_VAR
VAR_OUTPUT
END_VAR
VAR
END_VAR

END_FUNCTION_BLOCK

// HMI/POUs/Devices/Pumps/FB_HMI_PUMPS
FUNCTION_BLOCK FB_HMI_PUMPS EXTENDS FB_HMI_COMPONENT
VAR
	// System health & busy status
//    fbHealthStatus: 		FB_HMI_HEALTH_STATUS;
//    fbBusyStatus: 			FB_HMI_BUSY_STATUS;
//    fbStatusColor: 			T_HMI_COLORS;
	
	// Pumps
	fbRpBranchAButton: 		FB_HMI_BUTTON('RP A' , '', 	E_HMI_PUMPS_TABS.RP_BRANCH_A);
	fbRpBranchBButton: 		FB_HMI_BUTTON('RP B' , '', 	E_HMI_PUMPS_TABS.RP_BRANCH_B);
	fbTpBranchAButton: 		FB_HMI_BUTTON('TP A' , '', 	E_HMI_PUMPS_TABS.TP_BRANCH_A);
	fbTpBranchBButton: 		FB_HMI_BUTTON('TP B' , '', 	E_HMI_PUMPS_TABS.TP_BRANCH_B);
	
		// Pumps
	fbRpBranchA:			FB_HMI_RP_BRANCH_A;
	fbRpBranchB:			FB_HMI_RP_BRANCH_B;
	fbTpBranchA:			FB_HMI_TP_BRANCH_A;
	fbTpBranchB:			FB_HMI_TP_BRANCH_B;
	
	    // active tab of the main frame
    eActiveTab : E_HMI_PUMPS_TABS := E_HMI_PUMPS_TABS.RP_BRANCH_A;
    sActiveName : STRING;

END_VAR


// Pumps
 			
fbRpBranchA();
fbRpBranchB();
fbTpBranchA();
fbTpBranchB();

// Pumps

fbRpBranchAButton(stColor:= fbRpBranchA.fbStatusColor, nActiveTab:= eActiveTab, sActiveName:= sActiveName); 		
fbRpBranchBButton(stColor:= fbRpBranchB.fbStatusColor, nActiveTab:= eActiveTab, sActiveName:= sActiveName); 
fbTpBranchAButton(stColor:= fbTpBranchA.fbStatusColor, nActiveTab:= eActiveTab, sActiveName:= sActiveName); 
fbTpBranchBButton(stColor:= fbTpBranchB.fbStatusColor, nActiveTab:= eActiveTab, sActiveName:= sActiveName);

END_FUNCTION_BLOCK

// HMI/POUs/Util/Button/FB_HMI_BUTTON
FUNCTION_BLOCK FB_HMI_BUTTON
VAR_INPUT
    stColor : T_HMI_COLORS;
END_VAR
VAR_IN_OUT
    nActiveTab : INT;
    sActiveName : STRING;
END_VAR
VAR_OUTPUT
    sName : STRING;
    sIconName : STRING;
    nThisTab : INT;
    bActivated : BOOL;
    bNotActivated : BOOL;
    
    bIsNotGreen : BOOL;
    bIsNotRed : BOOL;
    bIsNotBlue : BOOL;
    bIsNotOrange : BOOL;
    bIsNotGray : BOOL;
END_VAR
VAR
    bDoActivate : BOOL;
    bPreviouslyActive : BOOL;
END_VAR

IF bDoActivate THEN
    nActiveTab := nThisTab;
    bDoActivate := FALSE;
END_IF

bActivated := nActiveTab = nThisTab;
bNotActivated := NOT bActivated;

IF bActivated AND NOT bPreviouslyActive THEN
    sActiveName := sName;
    bPreviouslyActive := TRUE;
END_IF

IF bNotActivated THEN
    bPreviouslyActive := FALSE;
END_IF

bIsNotRed    := stColor.bg <> E_HMI_Colors.RED;
bIsNotBlue   := stColor.bg <> E_HMI_Colors.BLUE;
bIsNotOrange := stColor.bg <> E_HMI_Colors.ORANGE;
bIsNotGray   := stColor.bg <> E_HMI_Colors.GRAY;
bIsNotGreen  := stColor.bg <> E_HMI_Colors.GREEN;

METHOD FB_init : BOOL
VAR_INPUT
	bInitRetains : BOOL; // if TRUE, the retain variables are initialized (warm start / cold start)
	bInCopyCode : BOOL;  // if TRUE, the instance afterwards gets moved into the copy code (online change)
    sName : STRING;
    sIconName : STRING;
    nThisTab : INT;
END_VAR
THIS^.sName := sName;
THIS^.sIconName := sIconName;
THIS^.nThisTab := nThisTab;
END_METHOD

METHOD M_SetIconName
VAR_INPUT
    sIconName : STRING;
END_VAR
THIS^.sIconName := sIconName;
END_METHOD

END_FUNCTION_BLOCK

// HMI/POUs/Devices/Pumps/FB_HMI_RP_BRANCH_A
FUNCTION_BLOCK FB_HMI_RP_BRANCH_A EXTENDS FB_HMI_COMPONENT
VAR_INPUT
END_VAR
VAR_OUTPUT
END_VAR
VAR
END_VAR

END_FUNCTION_BLOCK

// HMI/POUs/Devices/Pumps/FB_HMI_RP_BRANCH_B
FUNCTION_BLOCK FB_HMI_RP_BRANCH_B EXTENDS FB_HMI_COMPONENT
VAR_INPUT
END_VAR
VAR_OUTPUT
END_VAR
VAR
END_VAR

END_FUNCTION_BLOCK

// HMI/POUs/Devices/Pumps/FB_HMI_TP_BRANCH_A
FUNCTION_BLOCK FB_HMI_TP_BRANCH_A EXTENDS FB_HMI_COMPONENT
VAR_INPUT
END_VAR
VAR_OUTPUT
END_VAR
VAR
END_VAR

END_FUNCTION_BLOCK

// HMI/POUs/Devices/Pumps/FB_HMI_TP_BRANCH_B
FUNCTION_BLOCK FB_HMI_TP_BRANCH_B EXTENDS FB_HMI_COMPONENT
VAR_INPUT
END_VAR
VAR_OUTPUT
END_VAR
VAR
END_VAR

END_FUNCTION_BLOCK

// HMI/POUs/Devices/RH/FB_HMI_METIS_RH_SENSOR
FUNCTION_BLOCK FB_HMI_METIS_RH_SENSOR EXTENDS FB_HMI_COMPONENT
VAR_INPUT
END_VAR
VAR_OUTPUT
END_VAR
VAR_IN_OUT
    fbInstance : FB_METIS_RH_SENSOR;
END_VAR
VAR
END_VAR

fbHealthStatus(
    bIsEnabled := fbInstance.stat.bValid,
    bIsGood := NOT fbInstance.stat.bError);

fbBusyStatus(
    bIsEnabled := FALSE,
    bIsBusy := FALSE);

M_UpdateStatusColor();

END_FUNCTION_BLOCK

// HMI/POUs/Devices/Temperatures/Components/FB_HMI_TEMP_VOTERS
FUNCTION_BLOCK FB_HMI_TEMP_VOTERS EXTENDS FB_HMI_COMPONENT
VAR_INPUT
END_VAR
VAR_OUTPUT
END_VAR
VAR_IN_OUT
    fbInstance : FB_METIS_VOTERS;
END_VAR
VAR
    eActiveTab : E_HMI_VOTER_TABS;
    sActiveName : STRING;
    
    fbVoter1Button  : FB_HMI_BUTTON(sName := 'Master' , sIconName := '', nThisTab := E_HMI_VOTER_TABS.VOTER_1);
    fbVoter2Button  : FB_HMI_BUTTON(sName := 'Vot Master 1' , sIconName := '', nThisTab := E_HMI_VOTER_TABS.VOTER_2);
    fbVoter3Button  : FB_HMI_BUTTON(sName := 'Vot Master 2' , sIconName := '', nThisTab := E_HMI_VOTER_TABS.VOTER_3);
    
    
    fbVoter1 : FB_HMI_VOTER;
    fbVoter2 : FB_HMI_VOTER;
    fbVoter3 : FB_HMI_VOTER;
    
END_VAR

fbVoter1(fbInstance := fbInstance.vote_cry_1);
fbVoter2(fbInstance := fbInstance.vote_cry_2);
fbVoter3(fbInstance := fbInstance.vote_cry_3);


fbVoter1Button(stColor := fbVoter1.fbStatusColor, nActiveTab := eActiveTab, sActiveName := sActiveName);
fbVoter2Button(stColor := fbVoter2.fbStatusColor, nActiveTab := eActiveTab, sActiveName := sActiveName);
fbVoter3Button(stColor := fbVoter3.fbStatusColor, nActiveTab := eActiveTab, sActiveName := sActiveName);


fbHealthStatus(
    bIsEnabled :=  fbVoter1.fbHealthStatus.bEnabled
                OR fbVoter2.fbHealthStatus.bEnabled
                OR fbVoter3.fbHealthStatus.bEnabled,
    bIsGood :=  (fbVoter1.fbHealthStatus.bGood OR NOT fbVoter1.fbHealthStatus.bEnabled)
            AND (fbVoter2.fbHealthStatus.bGood OR NOT fbVoter2.fbHealthStatus.bEnabled)
            AND (fbVoter3.fbHealthStatus.bGood OR NOT fbVoter3.fbHealthStatus.bEnabled));

fbBusyStatus(bIsEnabled := FALSE);

M_UpdateStatusColor();

END_FUNCTION_BLOCK

// HMI/POUs/Devices/Voters/FB_HMI_VOTER
FUNCTION_BLOCK FB_HMI_VOTER EXTENDS FB_HMI_COMPONENT
VAR_INPUT
END_VAR
VAR_OUTPUT
END_VAR
VAR_IN_OUT
    fbInstance : FB_METIS_VOTER;
END_VAR
VAR
END_VAR

fbHealthStatus(
    bIsEnabled := fbInstance.stat.bEnabled,
    bIsGood := fbInstance.stat.bValid);
                     
fbBusyStatus(
    bIsEnabled := FALSE,
    bIsBusy := FALSE);

M_UpdateStatusColor();

END_FUNCTION_BLOCK

// HMI/POUs/Devices/Temperatures/FB_HMI_TEMPERATURES
FUNCTION_BLOCK FB_HMI_TEMPERATURES EXTENDS FB_HMI_COMPONENT
VAR_INPUT
END_VAR
VAR_OUTPUT
END_VAR

VAR_IN_OUT
    voters          : FB_METIS_VOTERS;
END_VAR
VAR
    // active tab of the main frame
    eActiveTab : E_HMI_TEMP_TABS := E_HMI_TEMP_TABS.VOTERS;
    sActiveName : STRING;
    
    // components
    fbVoters       		: FB_HMI_TEMP_VOTERS;

    
    // buttons
    fbVotersButton       : FB_HMI_BUTTON(sName := 'Voters'               , sIconName := '', nThisTab := E_HMI_CRY_TABS.VOTERS);

END_VAR

// update the components

fbVoters(fbInstance := voters);

// update the buttons

fbVotersButton(
    stColor     := fbVoters.fbStatusColor,
    nActiveTab  := eActiveTab,
    sActiveName := sActiveName);



// update the summary health/busy status
fbHealthStatus(
    bIsEnabled  := TRUE,
    bIsGood     :=     fbVoters.fbHealthStatus.bGood,
    bHasWarning :=     fbVoters.fbHealthStatus.bWarning);

fbBusyStatus(
    bIsEnabled   := TRUE,
    bIsBusy      :=    fbVoters.fbBusyStatus.bBusy);

M_UpdateStatusColor();

END_FUNCTION_BLOCK

// HMI/POUs/Devices/Valves/FB_HMI_VALVES
FUNCTION_BLOCK FB_HMI_VALVES EXTENDS FB_HMI_COMPONENT
VAR_INPUT
END_VAR
VAR_OUTPUT
END_VAR
VAR
END_VAR

END_FUNCTION_BLOCK

// HMI/POUs/Devices/FB_HMI_DEVICES
FUNCTION_BLOCK FB_HMI_DEVICES EXTENDS FB_HMI_COMPONENT
VAR_INPUT
END_VAR
VAR_OUTPUT
END_VAR
VAR
END_VAR

END_FUNCTION_BLOCK

// HMI/POUs/Events/FB_HMI_EVENTS
FUNCTION_BLOCK FB_HMI_EVENTS EXTENDS FB_HMI_COMPONENT
VAR_INPUT
END_VAR
VAR_OUTPUT
END_VAR
VAR
END_VAR

END_FUNCTION_BLOCK

// HMI/POUs/ICS_Interlocks/FB_HMI_ICS_INTERLOCKS
FUNCTION_BLOCK FB_HMI_ICS_INTERLOCKS EXTENDS FB_HMI_COMPONENT
VAR_INPUT
END_VAR
VAR_OUTPUT
END_VAR
VAR
END_VAR

END_FUNCTION_BLOCK

// HMI/POUs/Services/Status/F_HMI_BUSY_TO_COLOR
FUNCTION F_HMI_BUSY_TO_COLOR : T_HMI_COLORS
VAR_IN_OUT
    fbBusyStatus : FB_HMI_BUSY_STATUS;
END_VAR
VAR_OUTPUT
END_VAR
VAR
END_VAR

IF fbBusyStatus.bIdle THEN
    F_HMI_BUSY_TO_COLOR.fg := E_HMI_COLORS.BLACK;
    F_HMI_BUSY_TO_COLOR.bg := E_HMI_COLORS.GREEN;
ELSIF fbBusyStatus.bBusy THEN
	F_HMI_BUSY_TO_COLOR.fg := E_HMI_COLORS.WHITE;
	F_HMI_BUSY_TO_COLOR.bg := E_HMI_COLORS.BLUE;
ELSE
	F_HMI_BUSY_TO_COLOR.fg := E_HMI_COLORS.BLACK;
	F_HMI_BUSY_TO_COLOR.bg := E_HMI_COLORS.GRAY;
END_IF

END_FUNCTION

// HMI/POUs/Services/Status/F_HMI_HEALTH_TO_COLOR
FUNCTION F_HMI_HEALTH_TO_COLOR : T_HMI_COLORS
VAR_IN_OUT
    fbHealthStatus : FB_HMI_HEALTH_STATUS;
END_VAR
VAR_OUTPUT
END_VAR
VAR
END_VAR

IF fbHealthStatus.bGood THEN
    F_HMI_HEALTH_TO_COLOR.fg := E_HMI_COLORS.BLACK;
    F_HMI_HEALTH_TO_COLOR.bg := E_HMI_COLORS.GREEN;
ELSIF fbHealthStatus.bBad THEN
	F_HMI_HEALTH_TO_COLOR.fg := E_HMI_COLORS.WHITE;
	F_HMI_HEALTH_TO_COLOR.bg := E_HMI_COLORS.RED;
ELSIF fbHealthStatus.bWarning THEN
	F_HMI_HEALTH_TO_COLOR.fg := E_HMI_COLORS.WHITE;
	F_HMI_HEALTH_TO_COLOR.bg := E_HMI_COLORS.ORANGE;
ELSE
	F_HMI_HEALTH_TO_COLOR.fg := E_HMI_COLORS.BLACK;
	F_HMI_HEALTH_TO_COLOR.bg := E_HMI_COLORS.GRAY;
END_IF

END_FUNCTION

// HMI/POUs/Services/Status/FB_HMI_STATUS
FUNCTION_BLOCK FB_HMI_STATUS
VAR_INPUT
	sText : STRING;
	stColor : T_HMI_COLORS;
END_VAR
VAR_OUTPUT
END_VAR
VAR_IN_OUT
END_VAR
VAR
END_VAR

END_FUNCTION_BLOCK

// HMI/POUs/Services/FB_HMI_SERVICES
FUNCTION_BLOCK FB_HMI_SERVICES EXTENDS FB_HMI_COMPONENT
VAR_INPUT
END_VAR
VAR_OUTPUT
END_VAR
VAR_IN_OUT
    fbInstance : FB_SERVICES;
END_VAR
VAR
    fbTime : FB_HMI_SERVICES_TIME;
END_VAR

fbTime(fbInstance := fbInstance.fbTime);

fbHealthStatus(
    bIsEnabled  := fbTime.fbHealthStatus.bEnabled,
    bIsGood     := fbTime.fbHealthStatus.bGood);
fbBusyStatus(
    bIsEnabled  := fbTime.fbBusyStatus.bEnabled,
    bIsBusy     := fbTime.fbBusyStatus.bBusy);

M_UpdateStatusColor();

END_FUNCTION_BLOCK

// HMI/POUs/Services/FB_HMI_SERVICES_TIME
FUNCTION_BLOCK FB_HMI_SERVICES_TIME EXTENDS FB_HMI_COMPONENT
VAR_INPUT
END_VAR
VAR_OUTPUT
END_VAR
VAR_IN_OUT
    fbInstance : FB_TIME;
END_VAR
VAR
    // because GUI_TEMPLATE_TIME is a large height,
    // and because scrolling doesn't seem to work (bug in TC HMI?),
    // we display the GUI_TEMPLATE_TIME twice, with an offset in between 
    nAbsoluteMovementY : INT := -495;
    
    sUtc : STRING;
END_VAR


// update the health & busy states
fbHealthStatus(
    bIsGood     := fbInstance.stat.signal.qos = E_TIME_SIGNAL_QOS.VALID,
    bIsEnabled  := fbInstance.stat.signal.status = E_TIME_SIGNAL_STATUS.CONNECTED);
fbBusyStatus(bIsBusy := FALSE); // never busy

sUtc := LEFT(fbInstance.stat.sUtcTime, 19); 

M_UpdateStatusColor();

END_FUNCTION_BLOCK

// HMI/POUs/Subsystems/CFO/Components/FB_HMI_CFO_HEATERS
FUNCTION_BLOCK FB_HMI_CFO_HEATERS EXTENDS FB_HMI_COMPONENT
VAR_INPUT
END_VAR
VAR_OUTPUT
END_VAR
VAR_IN_OUT
    fbInstance : FB_METIS_HEATERS;
END_VAR
VAR
//    eActiveTab : E_HMI_CRY_HEATER_TABS;
//    sActiveName : STRING;
    
//    h_img_wuh_1_button  : FB_HMI_BUTTON(sName := 'H_IMG_WUH_1' , sIconName := '', nThisTab := E_HMI_IMG_HEATER_TABS.H_IMG_WUH_1);
//    h_img_wuh_2_button  : FB_HMI_BUTTON(sName := 'H_IMG_WUH_2' , sIconName := '', nThisTab := E_HMI_IMG_HEATER_TABS.H_IMG_WUH_2);
//    h_img_lmd_2_button  : FB_HMI_BUTTON(sName := 'H_IMG_LMD_2' , sIconName := '', nThisTab := E_HMI_IMG_HEATER_TABS.H_IMG_LMD_2);
//    h_img_lmp_2_button  : FB_HMI_BUTTON(sName := 'H_IMG_LMP_2' , sIconName := '', nThisTab := E_HMI_IMG_HEATER_TABS.H_IMG_LMP_2);
//    h_img_nd_2_button   : FB_HMI_BUTTON(sName := 'H_IMG_ND_2'  , sIconName := '', nThisTab := E_HMI_IMG_HEATER_TABS.H_IMG_ND_2);
    
//    h_img_wuh_1 : FB_HMI_METIS_HEATER;
//    h_img_wuh_2 : FB_HMI_METIS_HEATER;
//    h_img_lmd_2 : FB_HMI_METIS_HEATER;
//    h_img_lmp_2 : FB_HMI_METIS_HEATER;
//    h_img_nd_2  : FB_HMI_METIS_HEATER;
END_VAR

fbHealthStatus(bIsEnabled := FALSE);
fbBusyStatus(bIsEnabled := FALSE);

//fbHealthStatus(
//    bIsEnabled := TRUE,
//    bIsGood := NOT(    fbInstance.h_img_wuh_1.stat.bError
//                    OR fbInstance.h_img_wuh_2.stat.bError
//                    OR fbInstance.h_img_lmd_2.stat.bError
//                    OR fbInstance.h_img_lmp_2.stat.bError
//                    OR fbInstance.h_img_nd_2.stat.bError ),
//    bHasWarning := (    fbInstance.h_img_wuh_1.stat.bWarning
//                     OR fbInstance.h_img_wuh_2.stat.bWarning
//                     OR fbInstance.h_img_lmd_2.stat.bWarning
//                     OR fbInstance.h_img_lmp_2.stat.bWarning
//                     OR fbInstance.h_img_nd_2.stat.bWarning));

//fbBusyStatus(
//    bIsEnabled := TRUE,
//    bIsBusy := FALSE);

//h_img_wuh_1(fbInstance := fbInstance.h_img_wuh_1);
//h_img_wuh_2(fbInstance := fbInstance.h_img_wuh_2);
//h_img_lmd_2(fbInstance := fbInstance.h_img_lmd_2);
//h_img_lmp_2(fbInstance := fbInstance.h_img_lmp_2);
//h_img_nd_2(fbInstance := fbInstance.h_img_nd_2);

//h_img_wuh_1_button(stColor := h_img_wuh_1.fbStatusColor, nActiveTab := eActiveTab, sActiveName := sActiveName);
//h_img_wuh_2_button(stColor := h_img_wuh_2.fbStatusColor, nActiveTab := eActiveTab, sActiveName := sActiveName);
//h_img_lmd_2_button(stColor := h_img_lmd_2.fbStatusColor, nActiveTab := eActiveTab, sActiveName := sActiveName);
//h_img_lmp_2_button(stColor := h_img_lmp_2.fbStatusColor, nActiveTab := eActiveTab, sActiveName := sActiveName);
//h_img_nd_2_button(stColor := h_img_nd_2.fbStatusColor, nActiveTab := eActiveTab, sActiveName := sActiveName);

M_UpdateStatusColor();

END_FUNCTION_BLOCK

// HMI/POUs/Subsystems/CFO/Components/FB_HMI_CFO_TCTRL
FUNCTION_BLOCK FB_HMI_CFO_TCTRL EXTENDS FB_HMI_COMPONENT
VAR_INPUT
END_VAR
VAR_OUTPUT
END_VAR
VAR_IN_OUT
    fbInstance : FB_METIS_TCTRL;
END_VAR
VAR
//    eActiveTab : E_HMI_IMG_TC_TABS;
//    sActiveName : STRING;
    
//    tc_img_wuh_1_button  : FB_HMI_BUTTON(sName := 'TC_IMG_WUH_1' , sIconName := '', nThisTab := E_HMI_IMG_TC_TABS.TC_IMG_WUH_1);
//    tc_img_wuh_2_button  : FB_HMI_BUTTON(sName := 'TC_IMG_WUH_2' , sIconName := '', nThisTab := E_HMI_IMG_TC_TABS.TC_IMG_WUH_2);
//    tc_img_lmd_2_button  : FB_HMI_BUTTON(sName := 'TC_IMG_LMD_2' , sIconName := '', nThisTab := E_HMI_IMG_TC_TABS.TC_IMG_LMD_2);
//    tc_img_lmp_2_button  : FB_HMI_BUTTON(sName := 'TC_IMG_LMP_2' , sIconName := '', nThisTab := E_HMI_IMG_TC_TABS.TC_IMG_LMP_2);
//    tc_img_nd_2_button   : FB_HMI_BUTTON(sName := 'TC_IMG_ND_2'  , sIconName := '', nThisTab := E_HMI_IMG_TC_TABS.TC_IMG_ND_2);
    
//    tc_img_wuh_1 : FB_HMI_METIS_CTRL_DT670;
//    tc_img_wuh_2 : FB_HMI_METIS_CTRL_DT670;
//    tc_img_lmd_2 : FB_HMI_METIS_CTRL_DT670;
//    tc_img_lmp_2 : FB_HMI_METIS_CTRL_DT670;
//    tc_img_nd_2  : FB_HMI_METIS_CTRL_DT670;
END_VAR

fbHealthStatus(bIsEnabled := FALSE);
fbBusyStatus(bIsEnabled := FALSE);

//fbHealthStatus(
//    bIsEnabled := TRUE,
//    bIsGood := NOT(    fbInstance.tc_img_wuh_1.stat.bError
//                    OR fbInstance.tc_img_wuh_2.stat.bError
//                    OR fbInstance.tc_img_lmd_2.stat.bError
//                    OR fbInstance.tc_img_lmp_2.stat.bError
//                    OR fbInstance.tc_img_nd_2.stat.bError ),
//    bHasWarning := (    fbInstance.tc_img_wuh_1.stat.bWarning
//                     OR fbInstance.tc_img_wuh_2.stat.bWarning
//                     OR fbInstance.tc_img_lmd_2.stat.bWarning
//                     OR fbInstance.tc_img_lmp_2.stat.bWarning
//                     OR fbInstance.tc_img_nd_2.stat.bWarning));

//tc_img_wuh_1(fbInstance := fbInstance.tc_img_wuh_1);
//tc_img_wuh_2(fbInstance := fbInstance.tc_img_wuh_2);
//tc_img_lmd_2(fbInstance := fbInstance.tc_img_lmd_2);
//tc_img_lmp_2(fbInstance := fbInstance.tc_img_lmp_2);
//tc_img_nd_2(fbInstance := fbInstance.tc_img_nd_2);

//tc_img_wuh_1_button(stColor := tc_img_wuh_1.fbStatusColor, nActiveTab := eActiveTab, sActiveName := sActiveName);
//tc_img_wuh_2_button(stColor := tc_img_wuh_2.fbStatusColor, nActiveTab := eActiveTab, sActiveName := sActiveName);
//tc_img_lmd_2_button(stColor := tc_img_lmd_2.fbStatusColor, nActiveTab := eActiveTab, sActiveName := sActiveName);
//tc_img_lmp_2_button(stColor := tc_img_lmp_2.fbStatusColor, nActiveTab := eActiveTab, sActiveName := sActiveName);
//tc_img_nd_2_button(stColor := tc_img_nd_2.fbStatusColor, nActiveTab := eActiveTab, sActiveName := sActiveName);

//fbBusyStatus(
//    bIsEnabled := TRUE,
//    bIsBusy := FALSE);

M_UpdateStatusColor();

END_FUNCTION_BLOCK

// HMI/POUs/Subsystems/CFO/Components/FB_HMI_CFO_TEMPERATURES
FUNCTION_BLOCK FB_HMI_CFO_TEMPERATURES EXTENDS FB_HMI_COMPONENT
VAR_INPUT
END_VAR
VAR_OUTPUT
END_VAR
VAR_IN_OUT
    fbInstance : FB_METIS_TEMPERATURES;
END_VAR
VAR
END_VAR

fbHealthStatus(bIsEnabled := FALSE);
fbBusyStatus(bIsEnabled := FALSE);

//fbHealthStatus(
//    bIsEnabled := TRUE,
//    bIsGood :=     fbInstance.t_img_lpw_1.stat.bValid
//               AND fbInstance.t_img_lpw_2.stat.bValid
//               AND fbInstance.t_img_lfw_1.stat.bValid
//               AND fbInstance.t_img_lfw_2.stat.bValid
//               AND fbInstance.t_img_lpr_1.stat.bValid
//               AND fbInstance.t_img_bwu_3.stat.bValid
//               AND fbInstance.t_img_lnd_1.stat.bValid
//               AND fbInstance.t_img_lnd_2.stat.bValid
//               AND fbInstance.t_img_npw_1.stat.bValid
//               AND fbInstance.t_img_npw_2.stat.bValid
//               AND fbInstance.t_img_nfw_1.stat.bValid
//               AND fbInstance.t_img_nfw_2.stat.bValid
//               AND fbInstance.t_img_npr_1.stat.bValid
//               AND fbInstance.t_img_bwu_2.stat.bValid
//               AND fbInstance.t_img_nnd_1.stat.bValid
//               AND fbInstance.t_img_nnd_2.stat.bValid
//               AND fbInstance.t_img_opt_1.stat.bValid
//               AND fbInstance.t_img_bwu_1.stat.bValid
//               AND fbInstance.t_img_ctr_1.stat.bValid
//               AND fbInstance.t_img_ctr_2.stat.bValid
//               AND fbInstance.t_img_70k_1.stat.bValid
//               AND fbInstance.t_img_ln2_1.stat.bValid
//               AND fbInstance.t_img_ln2_2.stat.bValid
//               AND fbInstance.t_img_hex_1.stat.bValid
//               AND fbInstance.t_img_lmd_1.stat.bValid
//               AND fbInstance.t_img_lmd_2.stat.bValid
//               AND fbInstance.t_img_lmp_1.stat.bValid
//               AND fbInstance.t_img_lmp_2.stat.bValid
//               AND fbInstance.t_img_nd_1.stat.bValid
//               AND fbInstance.t_img_nd_2.stat.bValid,
//    bHasWarning := (    fbInstance.t_img_lpw_1.stat.bWarning
//                     OR fbInstance.t_img_lpw_2.stat.bWarning
//                     OR fbInstance.t_img_lfw_1.stat.bWarning
//                     OR fbInstance.t_img_lfw_2.stat.bWarning
//                     OR fbInstance.t_img_lpr_1.stat.bWarning
//                     OR fbInstance.t_img_bwu_3.stat.bWarning
//                     OR fbInstance.t_img_lnd_1.stat.bWarning
//                     OR fbInstance.t_img_lnd_2.stat.bWarning
//                     OR fbInstance.t_img_npw_1.stat.bWarning
//                     OR fbInstance.t_img_npw_2.stat.bWarning
//                     OR fbInstance.t_img_nfw_1.stat.bWarning
//                     OR fbInstance.t_img_nfw_2.stat.bWarning
//                     OR fbInstance.t_img_npr_1.stat.bWarning
//                     OR fbInstance.t_img_bwu_2.stat.bWarning
//                     OR fbInstance.t_img_nnd_1.stat.bWarning
//                     OR fbInstance.t_img_nnd_2.stat.bWarning
//                     OR fbInstance.t_img_opt_1.stat.bWarning
//                     OR fbInstance.t_img_bwu_1.stat.bWarning
//                     OR fbInstance.t_img_ctr_1.stat.bWarning
//                     OR fbInstance.t_img_ctr_2.stat.bWarning
//                     OR fbInstance.t_img_ln2_1.stat.bWarning
//                     OR fbInstance.t_img_ln2_1.stat.bWarning
//                     OR fbInstance.t_img_ln2_2.stat.bWarning
//                     OR fbInstance.t_img_hex_1.stat.bWarning
//                     OR fbInstance.t_img_lmd_1.stat.bWarning
//                     OR fbInstance.t_img_lmd_2.stat.bWarning
//                     OR fbInstance.t_img_lmp_1.stat.bWarning
//                     OR fbInstance.t_img_lmp_2.stat.bWarning
//                     OR fbInstance.t_img_nd_1.stat.bWarning
//                     OR fbInstance.t_img_nd_2.stat.bWarning));
                     
//fbBusyStatus(
//    bIsEnabled := TRUE,
//    bIsBusy := FALSE);

M_UpdateStatusColor();

END_FUNCTION_BLOCK

// HMI/POUs/Subsystems/CFO/Components/FB_HMI_CFO_VOTERS
FUNCTION_BLOCK FB_HMI_CFO_VOTERS EXTENDS FB_HMI_COMPONENT
VAR_INPUT
END_VAR
VAR_OUTPUT
END_VAR
VAR_IN_OUT
    fbInstance : FB_METIS_VOTERS;
END_VAR
VAR
    eActiveTab : E_HMI_VOTER_TABS;
    sActiveName : STRING;
    
    fbVoter1Button  : FB_HMI_BUTTON(sName := 'Voter 1' , sIconName := '', nThisTab := E_HMI_VOTER_TABS.VOTER_1);
    fbVoter2Button  : FB_HMI_BUTTON(sName := 'Voter 2' , sIconName := '', nThisTab := E_HMI_VOTER_TABS.VOTER_2);
    fbVoter3Button  : FB_HMI_BUTTON(sName := 'Voter 3' , sIconName := '', nThisTab := E_HMI_VOTER_TABS.VOTER_3);
    fbVoter4Button  : FB_HMI_BUTTON(sName := 'Voter 4' , sIconName := '', nThisTab := E_HMI_VOTER_TABS.VOTER_4);
    fbVoter5Button  : FB_HMI_BUTTON(sName := 'Voter 5' , sIconName := '', nThisTab := E_HMI_VOTER_TABS.VOTER_5);
    fbVoter6Button  : FB_HMI_BUTTON(sName := 'Voter 6' , sIconName := '', nThisTab := E_HMI_VOTER_TABS.VOTER_6);
    fbVoter7Button  : FB_HMI_BUTTON(sName := 'Voter 7' , sIconName := '', nThisTab := E_HMI_VOTER_TABS.VOTER_7);
    fbVoter8Button  : FB_HMI_BUTTON(sName := 'Voter 8' , sIconName := '', nThisTab := E_HMI_VOTER_TABS.VOTER_8);
    fbVoter9Button  : FB_HMI_BUTTON(sName := 'Voter 9' , sIconName := '', nThisTab := E_HMI_VOTER_TABS.VOTER_9);
    fbVoter10Button : FB_HMI_BUTTON(sName := 'Voter 10', sIconName := '', nThisTab := E_HMI_VOTER_TABS.VOTER_10);
    
    fbVoter1 : FB_HMI_VOTER;
    fbVoter2 : FB_HMI_VOTER;
    fbVoter3 : FB_HMI_VOTER;
    fbVoter4 : FB_HMI_VOTER;
    fbVoter5 : FB_HMI_VOTER;
    fbVoter6 : FB_HMI_VOTER;
    fbVoter7 : FB_HMI_VOTER;
    fbVoter8 : FB_HMI_VOTER;
    fbVoter9 : FB_HMI_VOTER;
    fbVoter10 : FB_HMI_VOTER;
END_VAR

fbHealthStatus(bIsEnabled := FALSE);
fbBusyStatus(bIsEnabled := FALSE);

//fbHealthStatus(
//    bIsEnabled :=  fbVoter1.fbHealthStatus.bEnabled
//                OR fbVoter2.fbHealthStatus.bEnabled
//                OR fbVoter3.fbHealthStatus.bEnabled
//                OR fbVoter4.fbHealthStatus.bEnabled
//                OR fbVoter5.fbHealthStatus.bEnabled
//                OR fbVoter6.fbHealthStatus.bEnabled
//                OR fbVoter7.fbHealthStatus.bEnabled
//                OR fbVoter8.fbHealthStatus.bEnabled
//                OR fbVoter9.fbHealthStatus.bEnabled
//                OR fbVoter10.fbHealthStatus.bEnabled,
//    bIsGood :=  (fbVoter1.fbHealthStatus.bGood OR NOT fbVoter1.fbHealthStatus.bEnabled)
//            AND (fbVoter2.fbHealthStatus.bGood OR NOT fbVoter2.fbHealthStatus.bEnabled)
//            AND (fbVoter3.fbHealthStatus.bGood OR NOT fbVoter3.fbHealthStatus.bEnabled)
//            AND (fbVoter4.fbHealthStatus.bGood OR NOT fbVoter4.fbHealthStatus.bEnabled)
//            AND (fbVoter5.fbHealthStatus.bGood OR NOT fbVoter5.fbHealthStatus.bEnabled)
//            AND (fbVoter6.fbHealthStatus.bGood OR NOT fbVoter6.fbHealthStatus.bEnabled)
//            AND (fbVoter7.fbHealthStatus.bGood OR NOT fbVoter7.fbHealthStatus.bEnabled)
//            AND (fbVoter8.fbHealthStatus.bGood OR NOT fbVoter8.fbHealthStatus.bEnabled)
//            AND (fbVoter9.fbHealthStatus.bGood OR NOT fbVoter9.fbHealthStatus.bEnabled)
//            AND (fbVoter10.fbHealthStatus.bGood OR NOT fbVoter10.fbHealthStatus.bEnabled));

//fbBusyStatus(
//    bIsEnabled := TRUE,
//    bIsBusy := FALSE);

//fbVoter1(fbInstance := fbInstance.vote_img_1);
//fbVoter2(fbInstance := fbInstance.vote_img_2);
//fbVoter3(fbInstance := fbInstance.vote_img_3);
//fbVoter4(fbInstance := fbInstance.vote_img_4);
//fbVoter5(fbInstance := fbInstance.vote_img_5);
//fbVoter6(fbInstance := fbInstance.vote_img_6);
//fbVoter7(fbInstance := fbInstance.vote_img_7);
//fbVoter8(fbInstance := fbInstance.vote_img_8);
//fbVoter9(fbInstance := fbInstance.vote_img_9);
//fbVoter10(fbInstance := fbInstance.vote_img_10);

//fbVoter1Button(stColor := fbVoter1.fbStatusColor, nActiveTab := eActiveTab, sActiveName := sActiveName);
//fbVoter2Button(stColor := fbVoter2.fbStatusColor, nActiveTab := eActiveTab, sActiveName := sActiveName);
//fbVoter3Button(stColor := fbVoter3.fbStatusColor, nActiveTab := eActiveTab, sActiveName := sActiveName);
//fbVoter4Button(stColor := fbVoter4.fbStatusColor, nActiveTab := eActiveTab, sActiveName := sActiveName);
//fbVoter5Button(stColor := fbVoter5.fbStatusColor, nActiveTab := eActiveTab, sActiveName := sActiveName);
//fbVoter6Button(stColor := fbVoter6.fbStatusColor, nActiveTab := eActiveTab, sActiveName := sActiveName);
//fbVoter7Button(stColor := fbVoter7.fbStatusColor, nActiveTab := eActiveTab, sActiveName := sActiveName);
//fbVoter8Button(stColor := fbVoter8.fbStatusColor, nActiveTab := eActiveTab, sActiveName := sActiveName);
//fbVoter9Button(stColor := fbVoter9.fbStatusColor, nActiveTab := eActiveTab, sActiveName := sActiveName);
//fbVoter10Button(stColor := fbVoter10.fbStatusColor, nActiveTab := eActiveTab, sActiveName := sActiveName);
    
M_UpdateStatusColor();

END_FUNCTION_BLOCK

// HMI/POUs/Subsystems/CFO/FB_HMI_CFO
FUNCTION_BLOCK FB_HMI_CFO EXTENDS FB_HMI_COMPONENT
VAR_INPUT
END_VAR
VAR_OUTPUT
END_VAR
VAR_IN_OUT
    temperatures    : FB_METIS_TEMPERATURES;
    heaters         : FB_METIS_HEATERS;
    voters          : FB_METIS_VOTERS;
    tctrl           : FB_METIS_TCTRL;
END_VAR
VAR
    // active tab of the main frame
    eActiveTab : E_HMI_CFO_TABS := E_HMI_CFO_TABS.TEMPERATURES;
    sActiveName : STRING;
    
    // components
    fbTemperatures : FB_HMI_CFO_TEMPERATURES;
    fbVoters       : FB_HMI_CFO_VOTERS;
    fbTControl     : FB_HMI_CFO_TCTRL;
    fbHeaters      : FB_HMI_CFO_HEATERS;
    
    // buttons
    fbTemperaturesButton : FB_HMI_BUTTON(sName := 'Temperatures'         , sIconName := '', nThisTab := E_HMI_CFO_TABS.TEMPERATURES);
    fbVotersButton       : FB_HMI_BUTTON(sName := 'Voters'               , sIconName := '', nThisTab := E_HMI_CFO_TABS.VOTERS);
    fbHeatersButton      : FB_HMI_BUTTON(sName := 'Heaters'              , sIconName := '', nThisTab := E_HMI_CFO_TABS.HEATERS);
    fbTControlButton     : FB_HMI_BUTTON(sName := 'Control loops'        , sIconName := '', nThisTab := E_HMI_CFO_TABS.TCONTROL);
END_VAR

// update the components
fbTemperatures(fbInstance := temperatures);
fbVoters(fbInstance := voters);
fbTControl(fbInstance := tctrl);
fbHeaters(fbInstance := heaters);

// update the buttons
fbTemperaturesButton(
    stColor     := fbTemperatures.fbStatusColor,
    nActiveTab  := eActiveTab,
    sActiveName := sActiveName);
fbVotersButton(
    stColor     := fbVoters.fbStatusColor,
    nActiveTab  := eActiveTab,
    sActiveName := sActiveName);
fbHeatersButton(
    stColor     := fbHeaters.fbStatusColor,
    nActiveTab  := eActiveTab,
    sActiveName := sActiveName);
fbTControlButton(
    stColor     := fbTControl.fbStatusColor,
    nActiveTab  := eActiveTab,
    sActiveName := sActiveName);


// update the summary health/busy status
fbHealthStatus(
    bIsEnabled  := TRUE,
    bIsGood     :=     fbTemperatures.fbHealthStatus.bGood
                   AND fbVoters.fbHealthStatus.bGood
                   AND fbTControl.fbHealthStatus.bGood
                   AND fbHeaters.fbHealthStatus.bGood,
    bHasWarning :=     fbTemperatures.fbHealthStatus.bWarning
                    OR fbVoters.fbHealthStatus.bWarning
                    OR fbTControl.fbHealthStatus.bWarning
                    OR fbHeaters.fbHealthStatus.bWarning);

fbBusyStatus(
    bIsEnabled   := TRUE,
    bIsBusy      :=    fbTemperatures.fbBusyStatus.bBusy
                    OR fbVoters.fbBusyStatus.bBusy
                    OR fbTControl.fbBusyStatus.bBusy
                    OR fbHeaters.fbBusyStatus.bBusy);

M_UpdateStatusColor();

END_FUNCTION_BLOCK

// HMI/POUs/Subsystems/CRY/Components/FB_HMI_CRY_HEATERS
FUNCTION_BLOCK FB_HMI_CRY_HEATERS EXTENDS FB_HMI_COMPONENT
VAR_INPUT
END_VAR
VAR_OUTPUT
END_VAR
VAR_IN_OUT
    fbInstance : FB_METIS_HEATERS;
END_VAR
VAR
    eActiveTab : E_HMI_CRY_HEATER_TABS;
    sActiveName : STRING;
    
    h_cry_sha_button  : FB_HMI_BUTTON(sName := 'H_CRY_SHA' , sIconName := '', nThisTab := E_HMI_CRY_HEATER_TABS.H_CRY_SHA);
    h_cry_shb_button  : FB_HMI_BUTTON(sName := 'H_CRY_SHB' , sIconName := '', nThisTab := E_HMI_CRY_HEATER_TABS.H_CRY_SHB);
    h_cry_shc_button  : FB_HMI_BUTTON(sName := 'H_CRY_SHC' , sIconName := '', nThisTab := E_HMI_CRY_HEATER_TABS.H_CRY_SHC);
    h_cry_sp_button   : FB_HMI_BUTTON(sName := 'H_CRY_SP'  , sIconName := '', nThisTab := E_HMI_CRY_HEATER_TABS.H_CRY_SP);
    h_cry_pta_button  : FB_HMI_BUTTON(sName := 'H_CRY_PTA' , sIconName := '', nThisTab := E_HMI_CRY_HEATER_TABS.H_CRY_PTA);
    h_cry_ptb_button  : FB_HMI_BUTTON(sName := 'H_CRY_PTB' , sIconName := '', nThisTab := E_HMI_CRY_HEATER_TABS.H_CRY_PTB);
    h_cry_ptc_button  : FB_HMI_BUTTON(sName := 'H_CRY_PTC' , sIconName := '', nThisTab := E_HMI_CRY_HEATER_TABS.H_CRY_PTC);
    h_cry_wi_button   : FB_HMI_BUTTON(sName := 'H_CRY_WI'  , sIconName := '', nThisTab := E_HMI_CRY_HEATER_TABS.H_CRY_WI);
    
    h_cry_sha : FB_HMI_METIS_HEATER;
    h_cry_shb : FB_HMI_METIS_HEATER;
    h_cry_shc : FB_HMI_METIS_HEATER;
    h_cry_sp  : FB_HMI_METIS_HEATER;
    h_cry_pta : FB_HMI_METIS_HEATER;
    h_cry_ptb : FB_HMI_METIS_HEATER;
    h_cry_ptc : FB_HMI_METIS_HEATER;
    h_cry_wi  : FB_HMI_METIS_HEATER;
END_VAR

fbHealthStatus(
    bIsEnabled := TRUE,
    bIsGood := NOT(    fbInstance.h_cry_sha.stat.bError
                    OR fbInstance.h_cry_shb.stat.bError
                    OR fbInstance.h_cry_shc.stat.bError
                    OR fbInstance.h_cry_sp.stat.bError
                    OR fbInstance.h_cry_pta.stat.bError
                    OR fbInstance.h_cry_ptb.stat.bError
                    OR fbInstance.h_cry_ptc.stat.bError
                    OR fbInstance.h_cry_wi.stat.bError),
    bHasWarning := (    fbInstance.h_cry_sha.stat.bWarning
                     OR fbInstance.h_cry_shb.stat.bWarning
                     OR fbInstance.h_cry_shc.stat.bWarning
                     OR fbInstance.h_cry_sp.stat.bWarning
                     OR fbInstance.h_cry_pta.stat.bWarning
                     OR fbInstance.h_cry_ptb.stat.bWarning
                     OR fbInstance.h_cry_ptc.stat.bWarning
                     OR fbInstance.h_cry_wi.stat.bWarning));

fbBusyStatus(
    bIsEnabled := TRUE,
    bIsBusy := FALSE);

h_cry_sha(fbInstance := fbInstance.h_cry_sha);
h_cry_shb(fbInstance := fbInstance.h_cry_shb);
h_cry_shc(fbInstance := fbInstance.h_cry_shc);
h_cry_sp( fbInstance := fbInstance.h_cry_sp);
h_cry_pta(fbInstance := fbInstance.h_cry_pta);
h_cry_ptb(fbInstance := fbInstance.h_cry_ptb);
h_cry_ptc(fbInstance := fbInstance.h_cry_ptc);
h_cry_wi( fbInstance := fbInstance.h_cry_wi);

h_cry_sha_button(stColor := h_cry_sha.fbStatusColor, nActiveTab := eActiveTab, sActiveName := sActiveName);
h_cry_shb_button(stColor := h_cry_shb.fbStatusColor, nActiveTab := eActiveTab, sActiveName := sActiveName);
h_cry_shc_button(stColor := h_cry_shc.fbStatusColor, nActiveTab := eActiveTab, sActiveName := sActiveName);
h_cry_sp_button( stColor := h_cry_sp.fbStatusColor , nActiveTab := eActiveTab, sActiveName := sActiveName);
h_cry_pta_button(stColor := h_cry_pta.fbStatusColor, nActiveTab := eActiveTab, sActiveName := sActiveName);
h_cry_ptb_button(stColor := h_cry_ptb.fbStatusColor, nActiveTab := eActiveTab, sActiveName := sActiveName);
h_cry_ptc_button(stColor := h_cry_ptc.fbStatusColor, nActiveTab := eActiveTab, sActiveName := sActiveName);
h_cry_wi_button( stColor := h_cry_wi.fbStatusColor , nActiveTab := eActiveTab, sActiveName := sActiveName);

M_UpdateStatusColor();

END_FUNCTION_BLOCK

// HMI/POUs/Subsystems/CRY/Components/FB_HMI_CRY_LN2CTRL
FUNCTION_BLOCK FB_HMI_CRY_LN2CTRL EXTENDS FB_HMI_COMPONENT
VAR_INPUT
END_VAR
VAR_OUTPUT
END_VAR
VAR_IN_OUT
    fbInstance :  ARRAY [1..3] OF FB_METIS_CRYO_LN2_LEVEL_CTRL;
END_VAR
VAR
END_VAR

fbHealthStatus(
    bIsEnabled := TRUE,
    bIsGood := NOT fbInstance[1].bError OR NOT fbInstance[2].bError OR NOT fbInstance[3].bError);

fbBusyStatus(
    bIsEnabled := TRUE,
    bIsBusy := FALSE);

M_UpdateStatusColor();

END_FUNCTION_BLOCK

// HMI/POUs/Subsystems/CRY/Components/FB_HMI_CRY_RH
FUNCTION_BLOCK FB_HMI_CRY_RH EXTENDS FB_HMI_COMPONENT
VAR_INPUT
END_VAR
VAR_OUTPUT
END_VAR
VAR_IN_OUT
    fbInstance : FB_METIS_RH;
END_VAR
VAR
    rh_cry_wi : FB_HMI_METIS_RH_SENSOR;
END_VAR

fbHealthStatus(
    bIsEnabled := TRUE,
    bIsGood := NOT fbInstance.rh_cry_wi.stat.bError);

fbBusyStatus(
    bIsEnabled := TRUE,
    bIsBusy := FALSE);

M_UpdateStatusColor();

END_FUNCTION_BLOCK

// HMI/POUs/Subsystems/CRY/Components/FB_HMI_CRY_TCTRL
FUNCTION_BLOCK FB_HMI_CRY_TCTRL EXTENDS FB_HMI_COMPONENT
VAR_INPUT
END_VAR
VAR_OUTPUT
END_VAR
VAR_IN_OUT
    fbInstance : FB_METIS_TCTRL;
END_VAR
VAR
    eActiveTab : E_HMI_CRY_TC_TABS;
    sActiveName : STRING;
    
    tc_cry_sha_button  : FB_HMI_BUTTON(sName := 'TC_CRY_SHA' , sIconName := '', nThisTab := E_HMI_CRY_TC_TABS.TC_CRY_SHA);
    tc_cry_shb_button  : FB_HMI_BUTTON(sName := 'TC_CRY_SHB' , sIconName := '', nThisTab := E_HMI_CRY_TC_TABS.TC_CRY_SHB);
    tc_cry_shc_button  : FB_HMI_BUTTON(sName := 'TC_CRY_SHC' , sIconName := '', nThisTab := E_HMI_CRY_TC_TABS.TC_CRY_SHC);
    tc_cry_pt_button    : FB_HMI_BUTTON(sName := 'TC_CRY_PT' , sIconName := '', nThisTab := E_HMI_CRY_TC_TABS.TC_CRY_PT);
    tc_cry_wi_button   : FB_HMI_BUTTON(sName := 'TC_CRY_WI'  , sIconName := '', nThisTab := E_HMI_CRY_TC_TABS.TC_CRY_WI);
	tc_cry_sp_button   : FB_HMI_BUTTON(sName := 'TC_CRY_SP'  , sIconName := '', nThisTab := E_HMI_CRY_TC_TABS.TC_CRY_SP);
    
    tc_cry_sha : FB_HMI_METIS_CTRL_TEMPERATURE;
    tc_cry_shb : FB_HMI_METIS_CTRL_TEMPERATURE;
    tc_cry_shc : FB_HMI_METIS_CTRL_TEMPERATURE;
    tc_cry_pt : FB_HMI_METIS_CTRL_TEMPERATURE;
    tc_cry_wi  : FB_HMI_METIS_CTRL_TEMPERATURE;
	tc_cry_sp  : FB_HMI_METIS_CTRL_TEMPERATURE;
END_VAR

fbHealthStatus(
    bIsEnabled := TRUE,
    bIsGood := NOT(    fbInstance.tc_cry_sha.stat.bError
                    OR fbInstance.tc_cry_shb.stat.bError
                    OR fbInstance.tc_cry_shc.stat.bError
                    OR fbInstance.tc_cry_pt.stat.bError
                    OR fbInstance.tc_cry_wi.stat.bError 
					OR fbInstance.tc_cry_sp.stat.bError),
    bHasWarning := (    fbInstance.tc_cry_sha.stat.bWarning
                     OR fbInstance.tc_cry_shb.stat.bWarning
                     OR fbInstance.tc_cry_shc.stat.bWarning
                     OR fbInstance.tc_cry_pt.stat.bWarning
                     OR fbInstance.tc_cry_wi.stat.bWarning
					 OR fbInstance.tc_cry_sp.stat.bWarning));

tc_cry_sha(fbInstance := fbInstance.tc_cry_sha);
tc_cry_shb(fbInstance := fbInstance.tc_cry_shb);
tc_cry_shc(fbInstance := fbInstance.tc_cry_shc);
tc_cry_pt(fbInstance := fbInstance.tc_cry_pt);
tc_cry_wi(fbInstance  := fbInstance.tc_cry_wi);
tc_cry_sp(fbInstance  := fbInstance.tc_cry_sp);

tc_cry_sha_button(stColor := tc_cry_sha.fbStatusColor, nActiveTab := eActiveTab, sActiveName := sActiveName);
tc_cry_shb_button(stColor := tc_cry_shb.fbStatusColor, nActiveTab := eActiveTab, sActiveName := sActiveName);
tc_cry_shc_button(stColor := tc_cry_shc.fbStatusColor, nActiveTab := eActiveTab, sActiveName := sActiveName);
tc_cry_pt_button(stColor := tc_cry_pt.fbStatusColor, nActiveTab := eActiveTab, sActiveName := sActiveName);
tc_cry_wi_button( stColor := tc_cry_wi.fbStatusColor,  nActiveTab := eActiveTab, sActiveName := sActiveName);
tc_cry_sp_button( stColor := tc_cry_sp.fbStatusColor,  nActiveTab := eActiveTab, sActiveName := sActiveName);

fbBusyStatus(
    bIsEnabled := TRUE,
    bIsBusy := FALSE);

M_UpdateStatusColor();

END_FUNCTION_BLOCK

// HMI/POUs/Subsystems/CRY/Components/FB_HMI_CRY_TEMPERATURES
FUNCTION_BLOCK FB_HMI_CRY_TEMPERATURES EXTENDS FB_HMI_COMPONENT
VAR_INPUT
END_VAR
VAR_OUTPUT
END_VAR
VAR_IN_OUT
    fbInstance : FB_METIS_TEMPERATURES;
END_VAR
VAR
END_VAR

fbHealthStatus(
    bIsEnabled := TRUE,
    bIsGood :=     fbInstance.t_cry_sha_1.stat.bValid
               AND fbInstance.t_cry_sha_2.stat.bValid
               AND fbInstance.t_cry_sha_3.stat.bValid
               AND fbInstance.t_cry_sha_4.stat.bValid
               AND fbInstance.t_cry_shb_1.stat.bValid
               AND fbInstance.t_cry_shb_2.stat.bValid
               AND fbInstance.t_cry_shb_3.stat.bValid
               AND fbInstance.t_cry_shb_4.stat.bValid
               AND fbInstance.t_cry_shc_1.stat.bValid
               AND fbInstance.t_cry_shc_2.stat.bValid
               AND fbInstance.t_cry_shc_3.stat.bValid
               AND fbInstance.t_cry_shc_4.stat.bValid
               AND fbInstance.t_cry_pta_1.stat.bValid
               AND fbInstance.t_cry_pta_2.stat.bValid
               AND fbInstance.t_cry_pta_3.stat.bValid
               AND fbInstance.t_cry_ptb_1.stat.bValid
               AND fbInstance.t_cry_ptb_2.stat.bValid
               AND fbInstance.t_cry_ptb_3.stat.bValid
               AND fbInstance.t_cry_ptc_1.stat.bValid
               AND fbInstance.t_cry_ptc_2.stat.bValid
               AND fbInstance.t_cry_ptc_3.stat.bValid
               AND fbInstance.t_cry_sp_1.stat.bValid
               AND fbInstance.t_cry_sp_2.stat.bValid
               AND fbInstance.t_cry_pca.stat.bValid
               AND fbInstance.t_cry_pcb.stat.bValid
               AND fbInstance.t_cry_wim.stat.bValid
               AND fbInstance.t_cry_wia.stat.bValid,
    bHasWarning := (    fbInstance.t_cry_sha_1.stat.bWarning
                     OR fbInstance.t_cry_sha_2.stat.bWarning
                     OR fbInstance.t_cry_sha_3.stat.bWarning
                     OR fbInstance.t_cry_sha_4.stat.bWarning
                     OR fbInstance.t_cry_shb_1.stat.bWarning
                     OR fbInstance.t_cry_shb_2.stat.bWarning
                     OR fbInstance.t_cry_shb_3.stat.bWarning
                     OR fbInstance.t_cry_shb_4.stat.bWarning
                     OR fbInstance.t_cry_shc_1.stat.bWarning
                     OR fbInstance.t_cry_shc_2.stat.bWarning
                     OR fbInstance.t_cry_shc_3.stat.bWarning
                     OR fbInstance.t_cry_shc_4.stat.bWarning
                     OR fbInstance.t_cry_pta_1.stat.bWarning
                     OR fbInstance.t_cry_pta_2.stat.bWarning
                     OR fbInstance.t_cry_pta_3.stat.bWarning
                     OR fbInstance.t_cry_ptb_1.stat.bWarning
                     OR fbInstance.t_cry_ptb_2.stat.bWarning
                     OR fbInstance.t_cry_ptb_3.stat.bWarning
                     OR fbInstance.t_cry_ptc_1.stat.bWarning
                     OR fbInstance.t_cry_ptc_2.stat.bWarning
                     OR fbInstance.t_cry_ptc_3.stat.bWarning
                     OR fbInstance.t_cry_sp_1.stat.bWarning
                     OR fbInstance.t_cry_sp_2.stat.bWarning));
                     
fbBusyStatus(
    bIsEnabled := TRUE,
    bIsBusy := FALSE);

M_UpdateStatusColor();

END_FUNCTION_BLOCK

// HMI/POUs/Subsystems/CRY/Components/FB_HMI_CRY_VOTERS
FUNCTION_BLOCK FB_HMI_CRY_VOTERS EXTENDS FB_HMI_COMPONENT
VAR_INPUT
END_VAR
VAR_OUTPUT
END_VAR
VAR_IN_OUT
    fbInstance : FB_METIS_VOTERS;
END_VAR
VAR
    eActiveTab : E_HMI_VOTER_TABS;
    sActiveName : STRING;
    
    fbVoter1Button  : FB_HMI_BUTTON(sName := 'Voter 1' , sIconName := '', nThisTab := E_HMI_VOTER_TABS.VOTER_1);
    fbVoter2Button  : FB_HMI_BUTTON(sName := 'Voter 2' , sIconName := '', nThisTab := E_HMI_VOTER_TABS.VOTER_2);
    fbVoter3Button  : FB_HMI_BUTTON(sName := 'Voter 3' , sIconName := '', nThisTab := E_HMI_VOTER_TABS.VOTER_3);
    fbVoter4Button  : FB_HMI_BUTTON(sName := 'Voter 4' , sIconName := '', nThisTab := E_HMI_VOTER_TABS.VOTER_4);
    fbVoter5Button  : FB_HMI_BUTTON(sName := 'Voter 5' , sIconName := '', nThisTab := E_HMI_VOTER_TABS.VOTER_5);
    fbVoter6Button  : FB_HMI_BUTTON(sName := 'Voter 6' , sIconName := '', nThisTab := E_HMI_VOTER_TABS.VOTER_6);
    fbVoter7Button  : FB_HMI_BUTTON(sName := 'Voter 7' , sIconName := '', nThisTab := E_HMI_VOTER_TABS.VOTER_7);
    fbVoter8Button  : FB_HMI_BUTTON(sName := 'Voter 8' , sIconName := '', nThisTab := E_HMI_VOTER_TABS.VOTER_8);
    fbVoter9Button  : FB_HMI_BUTTON(sName := 'Voter 9' , sIconName := '', nThisTab := E_HMI_VOTER_TABS.VOTER_9);
    fbVoter10Button : FB_HMI_BUTTON(sName := 'Voter 10', sIconName := '', nThisTab := E_HMI_VOTER_TABS.VOTER_10);
    
    fbVoter1 : FB_HMI_VOTER;
    fbVoter2 : FB_HMI_VOTER;
    fbVoter3 : FB_HMI_VOTER;
    fbVoter4 : FB_HMI_VOTER;
    fbVoter5 : FB_HMI_VOTER;
    fbVoter6 : FB_HMI_VOTER;
    fbVoter7 : FB_HMI_VOTER;
    fbVoter8 : FB_HMI_VOTER;
    fbVoter9 : FB_HMI_VOTER;
    fbVoter10 : FB_HMI_VOTER;
END_VAR

fbVoter1(fbInstance := fbInstance.vote_cry_1);
fbVoter2(fbInstance := fbInstance.vote_cry_2);
fbVoter3(fbInstance := fbInstance.vote_cry_3);
fbVoter4(fbInstance := fbInstance.vote_cry_4);
fbVoter5(fbInstance := fbInstance.vote_cry_5);
fbVoter6(fbInstance := fbInstance.vote_cry_6);
fbVoter7(fbInstance := fbInstance.vote_cry_7);
fbVoter8(fbInstance := fbInstance.vote_cry_8);
fbVoter9(fbInstance := fbInstance.vote_cry_9);
fbVoter10(fbInstance := fbInstance.vote_cry_10);

fbVoter1Button(stColor := fbVoter1.fbStatusColor, nActiveTab := eActiveTab, sActiveName := sActiveName);
fbVoter2Button(stColor := fbVoter2.fbStatusColor, nActiveTab := eActiveTab, sActiveName := sActiveName);
fbVoter3Button(stColor := fbVoter3.fbStatusColor, nActiveTab := eActiveTab, sActiveName := sActiveName);
fbVoter4Button(stColor := fbVoter4.fbStatusColor, nActiveTab := eActiveTab, sActiveName := sActiveName);
fbVoter5Button(stColor := fbVoter5.fbStatusColor, nActiveTab := eActiveTab, sActiveName := sActiveName);
fbVoter6Button(stColor := fbVoter6.fbStatusColor, nActiveTab := eActiveTab, sActiveName := sActiveName);
fbVoter7Button(stColor := fbVoter7.fbStatusColor, nActiveTab := eActiveTab, sActiveName := sActiveName);
fbVoter8Button(stColor := fbVoter8.fbStatusColor, nActiveTab := eActiveTab, sActiveName := sActiveName);
fbVoter9Button(stColor := fbVoter9.fbStatusColor, nActiveTab := eActiveTab, sActiveName := sActiveName);
fbVoter10Button(stColor := fbVoter10.fbStatusColor, nActiveTab := eActiveTab, sActiveName := sActiveName);

fbHealthStatus(
    bIsEnabled :=  fbVoter1.fbHealthStatus.bEnabled
                OR fbVoter2.fbHealthStatus.bEnabled
                OR fbVoter3.fbHealthStatus.bEnabled
                OR fbVoter4.fbHealthStatus.bEnabled
                OR fbVoter5.fbHealthStatus.bEnabled
                OR fbVoter6.fbHealthStatus.bEnabled
                OR fbVoter7.fbHealthStatus.bEnabled
                OR fbVoter8.fbHealthStatus.bEnabled
                OR fbVoter9.fbHealthStatus.bEnabled
                OR fbVoter10.fbHealthStatus.bEnabled,
    bIsGood :=  (fbVoter1.fbHealthStatus.bGood OR NOT fbVoter1.fbHealthStatus.bEnabled)
            AND (fbVoter2.fbHealthStatus.bGood OR NOT fbVoter2.fbHealthStatus.bEnabled)
            AND (fbVoter3.fbHealthStatus.bGood OR NOT fbVoter3.fbHealthStatus.bEnabled)
            AND (fbVoter4.fbHealthStatus.bGood OR NOT fbVoter4.fbHealthStatus.bEnabled)
            AND (fbVoter5.fbHealthStatus.bGood OR NOT fbVoter5.fbHealthStatus.bEnabled)
            AND (fbVoter6.fbHealthStatus.bGood OR NOT fbVoter6.fbHealthStatus.bEnabled)
            AND (fbVoter7.fbHealthStatus.bGood OR NOT fbVoter7.fbHealthStatus.bEnabled)
            AND (fbVoter8.fbHealthStatus.bGood OR NOT fbVoter8.fbHealthStatus.bEnabled)
            AND (fbVoter9.fbHealthStatus.bGood OR NOT fbVoter9.fbHealthStatus.bEnabled)
            AND (fbVoter10.fbHealthStatus.bGood OR NOT fbVoter10.fbHealthStatus.bEnabled));

fbBusyStatus(bIsEnabled := FALSE);

M_UpdateStatusColor();

END_FUNCTION_BLOCK

// HMI/POUs/Subsystems/CRY/FB_HMI_CRY
FUNCTION_BLOCK FB_HMI_CRY EXTENDS FB_HMI_COMPONENT
VAR_INPUT
END_VAR
VAR_OUTPUT
END_VAR
VAR_IN_OUT
    temperatures    : FB_METIS_TEMPERATURES;
    rh              : FB_METIS_RH;
    heaters         : FB_METIS_HEATERS;
    voters          : FB_METIS_VOTERS;
    tctrl           : FB_METIS_TCTRL;
	ln2ctrl			: ARRAY [1..3] OF FB_METIS_CRYO_LN2_LEVEL_CTRL;
END_VAR
VAR
    // active tab of the main frame
    eActiveTab : E_HMI_CRY_TABS := E_HMI_CRY_TABS.TEMPERATURES;
    sActiveName : STRING;
    
    // components
    fbTemperatures 		: FB_HMI_CRY_TEMPERATURES;
    fbRh           		: FB_HMI_CRY_RH;
    fbVoters       		: FB_HMI_CRY_VOTERS;
    fbTControl     		: FB_HMI_CRY_TCTRL;
    fbHeaters      		: FB_HMI_CRY_HEATERS;
	fbLN2LevelControl   : FB_HMI_CRY_LN2CTRL;
    
    // buttons
    fbTemperaturesButton : FB_HMI_BUTTON(sName := 'Temperatures'         , sIconName := '', nThisTab := E_HMI_CRY_TABS.TEMPERATURES);
    fbRhButton           : FB_HMI_BUTTON(sName := 'Relative Humidity'    , sIconName := '', nThisTab := E_HMI_CRY_TABS.RH);
    fbVotersButton       : FB_HMI_BUTTON(sName := 'Voters'               , sIconName := '', nThisTab := E_HMI_CRY_TABS.VOTERS);
    fbHeatersButton      : FB_HMI_BUTTON(sName := 'Heaters'              , sIconName := '', nThisTab := E_HMI_CRY_TABS.HEATERS);
    fbTControlButton     : FB_HMI_BUTTON(sName := 'Control loops'        , sIconName := '', nThisTab := E_HMI_CRY_TABS.TCONTROL);
	fbLN2ControlButton   : FB_HMI_BUTTON(sName := 'LN2 Level Control'    , sIconName := '', nThisTab := E_HMI_CRY_TABS.LN2CONTROL);
END_VAR

// update the components
fbTemperatures(fbInstance := temperatures);
fbRh(fbInstance := rh);
fbVoters(fbInstance := voters);
fbTControl(fbInstance := tctrl);
fbHeaters(fbInstance := heaters);
fbLN2LevelControl(fbInstance := ln2ctrl);
// update the buttons
fbTemperaturesButton(
    stColor     := fbTemperatures.fbStatusColor,
    nActiveTab  := eActiveTab,
    sActiveName := sActiveName);
fbRhButton(
    stColor     := fbRh.fbStatusColor,
    nActiveTab  := eActiveTab,
    sActiveName := sActiveName);
fbVotersButton(
    stColor     := fbVoters.fbStatusColor,
    nActiveTab  := eActiveTab,
    sActiveName := sActiveName);
fbHeatersButton(
    stColor     := fbHeaters.fbStatusColor,
    nActiveTab  := eActiveTab,
    sActiveName := sActiveName);
fbTControlButton(
    stColor     := fbTControl.fbStatusColor,
    nActiveTab  := eActiveTab,
    sActiveName := sActiveName);
fbLN2ControlButton(
	stColor     := fbLN2LevelControl.fbStatusColor,
    nActiveTab  := eActiveTab,
    sActiveName := sActiveName);


// update the summary health/busy status
fbHealthStatus(
    bIsEnabled  := TRUE,
    bIsGood     :=     fbTemperatures.fbHealthStatus.bGood
                   AND fbRh.fbHealthStatus.bGood
                   AND fbVoters.fbHealthStatus.bGood
                   AND fbTControl.fbHealthStatus.bGood
                   AND fbHeaters.fbHealthStatus.bGood
				   AND fbLN2LevelControl.fbHealthStatus.bGood,
    bHasWarning :=     fbTemperatures.fbHealthStatus.bWarning
                    OR fbRh.fbHealthStatus.bGood
                    OR fbVoters.fbHealthStatus.bWarning
                    OR fbTControl.fbHealthStatus.bWarning
                    OR fbHeaters.fbHealthStatus.bWarning
					OR fbLN2LevelControl.fbHealthStatus.bWarning);

fbBusyStatus(
    bIsEnabled   := TRUE,
    bIsBusy      :=    fbTemperatures.fbBusyStatus.bBusy
                    OR fbRh.fbBusyStatus.bBusy
                    OR fbVoters.fbBusyStatus.bBusy
                    OR fbTControl.fbBusyStatus.bBusy
                    OR fbHeaters.fbBusyStatus.bBusy
					OR fbLN2LevelControl.fbBusyStatus.bBusy);

M_UpdateStatusColor();

END_FUNCTION_BLOCK

// HMI/POUs/Subsystems/ICS/FB_HMI_ICS
FUNCTION_BLOCK FB_HMI_ICS EXTENDS FB_HMI_COMPONENT
VAR_INPUT
END_VAR
VAR_OUTPUT
END_VAR
VAR_IN_OUT
	{attribute 'OPC.UA.DA' := '0'}
    ccus    : FB_METIS_CCUS;
END_VAR
VAR
    // active tab of the main frame
    eActiveTab : E_HMI_ICS_TABS := E_HMI_ICS_TABS.CCU_NS_2; // CHANGE to first available cabinet
    sActiveName : STRING;
    
    // components
    fbCCU_NS_1        : FB_HMI_CCU;
    fbCCU_NS_2        : FB_HMI_CCU;
    // fbCCU_NS_3        : FB_HMI_CCU;
    // fbCCU_NS_4        : FB_HMI_CCU;
    // fbCCU_NS_5        : FB_HMI_CCU;
    // fbCCU_NS_6        : FB_HMI_CCU;
    
    // buttons
    fbCCU_NS_1_Button    : FB_HMI_BUTTON(sName := 'CCU_NS_1', sIconName := '', nThisTab := E_HMI_ICS_TABS.CCU_NS_1);
    fbCCU_NS_2_Button    : FB_HMI_BUTTON(sName := 'CCU_NS_2', sIconName := '', nThisTab := E_HMI_ICS_TABS.CCU_NS_2);
    // add more buttons here
    fbConfigsButton : FB_HMI_BUTTON(sName := 'Configs'       , sIconName := '', nThisTab := E_HMI_ICS_TABS.CCU_CONFIGS);
    
    // configs color
    stConfigsColor : T_HMI_COLORS;
    fbConfigsHealthStatus : FB_HMI_HEALTH_STATUS;
    fbConfigsBusyStatus : FB_HMI_Busy_STATUS;
END_VAR

// update the components
fbCCU_NS_1(fbInstance := ccus.ccu_ns_1);
fbCCU_NS_2(fbInstance := ccus.ccu_ns_2);

M_UpdateConfigsColor(
    aCoolingConfig := ccus.aCoolingConfig, 
    aPowerConfig   := ccus.aPowerConfig);

// update the buttons
fbCCU_NS_1_Button(
    stColor     := fbCCU_NS_1.fbStatusColor,
    nActiveTab  := eActiveTab,
    sActiveName := sActiveName);
fbCCU_NS_2_Button(
    stColor     := fbCCU_NS_2.fbStatusColor,
    nActiveTab  := eActiveTab,
    sActiveName := sActiveName);
fbConfigsButton(
    stColor     := stConfigsColor,
    nActiveTab  := eActiveTab,
    sActiveName := sActiveName);
    

// update the summary health/busy status
fbHealthStatus(
    bIsEnabled  := TRUE,
    bIsGood     :=     fbCCU_NS_1.fbHealthStatus.bGood
                   AND fbCCU_NS_2.fbHealthStatus.bGood
                   AND fbConfigsHealthStatus.bGood,
    bHasWarning :=     fbCCU_NS_1.fbHealthStatus.bWarning
                    OR fbCCU_NS_2.fbHealthStatus.bWarning
                    OR fbConfigsHealthStatus.bWarning);

fbBusyStatus(
    bIsEnabled   := TRUE,
    bIsBusy      :=    fbCCU_NS_1.fbBusyStatus.bBusy
                    OR fbCCU_NS_2.fbBusyStatus.bBusy
                    OR fbConfigsBusyStatus.bBusy);

M_UpdateStatusColor();

METHOD M_UpdateConfigsColor
VAR_INPUT
END_VAR
VAR_IN_OUT
	{attribute 'OPC.UA.DA' := '0'}
    // cooling config handlers
    aCoolingConfig : ARRAY[1..2] OF FB_READ_WRITE_CAB_COOLING_CONFIG;
    
	{attribute 'OPC.UA.DA' := '0'}
    // power config handlers
    aPowerConfig : ARRAY[1..2] OF FB_READ_WRITE_CAB_POWER_CONFIG;
END_VAR
VAR
    i : INT;
    bAllGood : BOOL;
    bAnyBusy : BOOL;
END_VAR
bAllGood := TRUE;
bAnyBusy := FALSE;
FOR i := 1 TO 2 DO
    IF aCoolingConfig[i].bReadError OR aCoolingConfig[i].bWriteError
       OR aPowerConfig[i].bReadError OR aPowerConfig[i].bWriteError 
    THEN
        bAllGood := FALSE;
	END_IF
    IF aCoolingConfig[i].bReading OR aCoolingConfig[i].bWriting
       OR aPowerConfig[i].bReading OR aPowerConfig[i].bWriting 
    THEN
        bAnyBusy := TRUE;
	END_IF
END_FOR

fbConfigsHealthStatus(bIsEnabled := TRUE, bIsGood := bAllGood);
fbConfigsBusyStatus(bIsEnabled := TRUE, bIsBusy := bAnyBusy);

stConfigsColor := F_HMI_HEALTH_BUSY_TO_COLOR(
    fbConfigsHealthStatus, 
    fbConfigsBusyStatus);
END_METHOD

END_FUNCTION_BLOCK

// HMI/POUs/Subsystems/IMG/Components/FB_HMI_IMG_HEATERS
FUNCTION_BLOCK FB_HMI_IMG_HEATERS EXTENDS FB_HMI_COMPONENT
VAR_INPUT
    bConnected : BOOL;
END_VAR
VAR_OUTPUT
END_VAR
VAR_IN_OUT
    fbInstance : FB_METIS_HEATERS;
END_VAR
VAR
    eActiveTab : E_HMI_IMG_HEATER_TABS;
    sActiveName : STRING;
    
    h_img_wuh_1_button  : FB_HMI_BUTTON(sName := 'H_IMG_WUH_1' , sIconName := '', nThisTab := E_HMI_IMG_HEATER_TABS.H_IMG_WUH_1);
    h_img_wuh_2_button  : FB_HMI_BUTTON(sName := 'H_IMG_WUH_2' , sIconName := '', nThisTab := E_HMI_IMG_HEATER_TABS.H_IMG_WUH_2);
    h_img_lmd_2_button  : FB_HMI_BUTTON(sName := 'H_IMG_LMD_2' , sIconName := '', nThisTab := E_HMI_IMG_HEATER_TABS.H_IMG_LMD_2);
    h_img_lmp_2_button  : FB_HMI_BUTTON(sName := 'H_IMG_LMP_2' , sIconName := '', nThisTab := E_HMI_IMG_HEATER_TABS.H_IMG_LMP_2);
    h_img_nd_2_button   : FB_HMI_BUTTON(sName := 'H_IMG_ND_2'  , sIconName := '', nThisTab := E_HMI_IMG_HEATER_TABS.H_IMG_ND_2);
    
    h_img_wuh_1 : FB_HMI_METIS_HEATER;
    h_img_wuh_2 : FB_HMI_METIS_HEATER;
    h_img_lmd_2 : FB_HMI_METIS_HEATER;
    h_img_lmp_2 : FB_HMI_METIS_HEATER;
    h_img_nd_2  : FB_HMI_METIS_HEATER;
END_VAR

fbHealthStatus(
    bIsEnabled := bConnected,
    bIsGood := NOT(    fbInstance.h_img_wuh_1.stat.bError
                    OR fbInstance.h_img_wuh_2.stat.bError
                    OR fbInstance.h_img_lmd_2.stat.bError
                    OR fbInstance.h_img_lmp_2.stat.bError
                    OR fbInstance.h_img_nd_2.stat.bError ),
    bHasWarning := (    fbInstance.h_img_wuh_1.stat.bWarning
                     OR fbInstance.h_img_wuh_2.stat.bWarning
                     OR fbInstance.h_img_lmd_2.stat.bWarning
                     OR fbInstance.h_img_lmp_2.stat.bWarning
                     OR fbInstance.h_img_nd_2.stat.bWarning));

fbBusyStatus(
    bIsEnabled := bConnected,
    bIsBusy := FALSE);

h_img_wuh_1(fbInstance := fbInstance.h_img_wuh_1);
h_img_wuh_2(fbInstance := fbInstance.h_img_wuh_2);
h_img_lmd_2(fbInstance := fbInstance.h_img_lmd_2);
h_img_lmp_2(fbInstance := fbInstance.h_img_lmp_2);
h_img_nd_2(fbInstance := fbInstance.h_img_nd_2);

h_img_wuh_1_button(stColor := h_img_wuh_1.fbStatusColor, nActiveTab := eActiveTab, sActiveName := sActiveName);
h_img_wuh_2_button(stColor := h_img_wuh_2.fbStatusColor, nActiveTab := eActiveTab, sActiveName := sActiveName);
h_img_lmd_2_button(stColor := h_img_lmd_2.fbStatusColor, nActiveTab := eActiveTab, sActiveName := sActiveName);
h_img_lmp_2_button(stColor := h_img_lmp_2.fbStatusColor, nActiveTab := eActiveTab, sActiveName := sActiveName);
h_img_nd_2_button(stColor := h_img_nd_2.fbStatusColor, nActiveTab := eActiveTab, sActiveName := sActiveName);

M_UpdateStatusColor();

END_FUNCTION_BLOCK

// HMI/POUs/Subsystems/IMG/Components/FB_HMI_IMG_TCTRL
FUNCTION_BLOCK FB_HMI_IMG_TCTRL EXTENDS FB_HMI_COMPONENT
VAR_INPUT
    bConnected : BOOL;
END_VAR
VAR_OUTPUT
END_VAR
VAR_IN_OUT
    fbInstance : FB_METIS_TCTRL;
END_VAR
VAR
    eActiveTab : E_HMI_IMG_TC_TABS;
    sActiveName : STRING;
    
    tc_img_wuh_button    : FB_HMI_BUTTON(sName := 'TC_IMG_WUH'   , sIconName := '', nThisTab := E_HMI_IMG_TC_TABS.TC_IMG_WUH);
    tc_img_lmd_2_button  : FB_HMI_BUTTON(sName := 'TC_IMG_LMD_2' , sIconName := '', nThisTab := E_HMI_IMG_TC_TABS.TC_IMG_LMD_2);
    tc_img_lmp_2_button  : FB_HMI_BUTTON(sName := 'TC_IMG_LMP_2' , sIconName := '', nThisTab := E_HMI_IMG_TC_TABS.TC_IMG_LMP_2);
    tc_img_nd_2_button   : FB_HMI_BUTTON(sName := 'TC_IMG_ND_2'  , sIconName := '', nThisTab := E_HMI_IMG_TC_TABS.TC_IMG_ND_2);
    
    tc_img_wuh   : FB_HMI_METIS_CTRL_TEMPERATURE;
    tc_img_lmd_2 : FB_HMI_METIS_CTRL_TEMPERATURE;
    tc_img_lmp_2 : FB_HMI_METIS_CTRL_TEMPERATURE;
    tc_img_nd_2  : FB_HMI_METIS_CTRL_TEMPERATURE;
END_VAR

fbHealthStatus(
    bIsEnabled := bConnected,
    bIsGood := NOT(    fbInstance.tc_img_wuh.stat.bError
                    OR fbInstance.tc_img_lmd_2.stat.bError
                    OR fbInstance.tc_img_lmp_2.stat.bError
                    OR fbInstance.tc_img_nd_2.stat.bError ),
    bHasWarning := (    fbInstance.tc_img_wuh.stat.bWarning
                     OR fbInstance.tc_img_lmd_2.stat.bWarning
                     OR fbInstance.tc_img_lmp_2.stat.bWarning
                     OR fbInstance.tc_img_nd_2.stat.bWarning));

tc_img_wuh(fbInstance := fbInstance.tc_img_wuh);
tc_img_lmd_2(fbInstance := fbInstance.tc_img_lmd_2);
tc_img_lmp_2(fbInstance := fbInstance.tc_img_lmp_2);
tc_img_nd_2(fbInstance := fbInstance.tc_img_nd_2);

tc_img_wuh_button(stColor := tc_img_wuh.fbStatusColor, nActiveTab := eActiveTab, sActiveName := sActiveName);
tc_img_lmd_2_button(stColor := tc_img_lmd_2.fbStatusColor, nActiveTab := eActiveTab, sActiveName := sActiveName);
tc_img_lmp_2_button(stColor := tc_img_lmp_2.fbStatusColor, nActiveTab := eActiveTab, sActiveName := sActiveName);
tc_img_nd_2_button(stColor := tc_img_nd_2.fbStatusColor, nActiveTab := eActiveTab, sActiveName := sActiveName);

fbBusyStatus(
    bIsEnabled := bConnected,
    bIsBusy := FALSE);

M_UpdateStatusColor();

END_FUNCTION_BLOCK

// HMI/POUs/Subsystems/IMG/Components/FB_HMI_IMG_TEMPERATURES
FUNCTION_BLOCK FB_HMI_IMG_TEMPERATURES EXTENDS FB_HMI_COMPONENT
VAR_INPUT
    bConnected : BOOL;
END_VAR
VAR_OUTPUT
END_VAR
VAR_IN_OUT
    fbInstance : FB_METIS_TEMPERATURES;
END_VAR
VAR
END_VAR

fbHealthStatus(
    bIsEnabled := bConnected,
    bIsGood :=     fbInstance.t_img_lpw_1.stat.bValid
               AND fbInstance.t_img_lpw_2.stat.bValid
               AND fbInstance.t_img_lfw_1.stat.bValid
               AND fbInstance.t_img_lfw_2.stat.bValid
               AND fbInstance.t_img_lpr_1.stat.bValid
               AND fbInstance.t_img_bwu_3.stat.bValid
               AND fbInstance.t_img_lnd_1.stat.bValid
               AND fbInstance.t_img_lnd_2.stat.bValid
               AND fbInstance.t_img_npw_1.stat.bValid
               AND fbInstance.t_img_npw_2.stat.bValid
               AND fbInstance.t_img_nfw_1.stat.bValid
               AND fbInstance.t_img_nfw_2.stat.bValid
               AND fbInstance.t_img_npr_1.stat.bValid
               AND fbInstance.t_img_bwu_2.stat.bValid
               AND fbInstance.t_img_nnd_1.stat.bValid
               AND fbInstance.t_img_nnd_2.stat.bValid
               AND fbInstance.t_img_opt_1.stat.bValid
               AND fbInstance.t_img_bwu_1.stat.bValid
               AND fbInstance.t_img_ctr_1.stat.bValid
               AND fbInstance.t_img_ctr_2.stat.bValid
               AND fbInstance.t_img_70k_1.stat.bValid
               AND fbInstance.t_img_ln2_1.stat.bValid
               AND fbInstance.t_img_ln2_2.stat.bValid
               AND fbInstance.t_img_hex_1.stat.bValid
               AND fbInstance.t_img_lmd_1.stat.bValid
               AND fbInstance.t_img_lmd_2.stat.bValid
               AND fbInstance.t_img_lmp_1.stat.bValid
               AND fbInstance.t_img_lmp_2.stat.bValid
               AND fbInstance.t_img_nd_1.stat.bValid
               AND fbInstance.t_img_nd_2.stat.bValid,
    bHasWarning := (    fbInstance.t_img_lpw_1.stat.bWarning
                     OR fbInstance.t_img_lpw_2.stat.bWarning
                     OR fbInstance.t_img_lfw_1.stat.bWarning
                     OR fbInstance.t_img_lfw_2.stat.bWarning
                     OR fbInstance.t_img_lpr_1.stat.bWarning
                     OR fbInstance.t_img_bwu_3.stat.bWarning
                     OR fbInstance.t_img_lnd_1.stat.bWarning
                     OR fbInstance.t_img_lnd_2.stat.bWarning
                     OR fbInstance.t_img_npw_1.stat.bWarning
                     OR fbInstance.t_img_npw_2.stat.bWarning
                     OR fbInstance.t_img_nfw_1.stat.bWarning
                     OR fbInstance.t_img_nfw_2.stat.bWarning
                     OR fbInstance.t_img_npr_1.stat.bWarning
                     OR fbInstance.t_img_bwu_2.stat.bWarning
                     OR fbInstance.t_img_nnd_1.stat.bWarning
                     OR fbInstance.t_img_nnd_2.stat.bWarning
                     OR fbInstance.t_img_opt_1.stat.bWarning
                     OR fbInstance.t_img_bwu_1.stat.bWarning
                     OR fbInstance.t_img_ctr_1.stat.bWarning
                     OR fbInstance.t_img_ctr_2.stat.bWarning
                     OR fbInstance.t_img_ln2_1.stat.bWarning
                     OR fbInstance.t_img_ln2_1.stat.bWarning
                     OR fbInstance.t_img_ln2_2.stat.bWarning
                     OR fbInstance.t_img_hex_1.stat.bWarning
                     OR fbInstance.t_img_lmd_1.stat.bWarning
                     OR fbInstance.t_img_lmd_2.stat.bWarning
                     OR fbInstance.t_img_lmp_1.stat.bWarning
                     OR fbInstance.t_img_lmp_2.stat.bWarning
                     OR fbInstance.t_img_nd_1.stat.bWarning
                     OR fbInstance.t_img_nd_2.stat.bWarning));
                     
fbBusyStatus(
    bIsEnabled := bConnected,
    bIsBusy := FALSE);

M_UpdateStatusColor();

END_FUNCTION_BLOCK

// HMI/POUs/Subsystems/IMG/Components/FB_HMI_IMG_VOTERS
FUNCTION_BLOCK FB_HMI_IMG_VOTERS EXTENDS FB_HMI_COMPONENT
VAR_INPUT
    bConnected : BOOL;
END_VAR
VAR_OUTPUT
END_VAR
VAR_IN_OUT
    fbInstance : FB_METIS_VOTERS;
END_VAR
VAR
    eActiveTab : E_HMI_VOTER_TABS;
    sActiveName : STRING;
    
    fbVoter1Button  : FB_HMI_BUTTON(sName := 'Voter 1' , sIconName := '', nThisTab := E_HMI_VOTER_TABS.VOTER_1);
    fbVoter2Button  : FB_HMI_BUTTON(sName := 'Voter 2' , sIconName := '', nThisTab := E_HMI_VOTER_TABS.VOTER_2);
    fbVoter3Button  : FB_HMI_BUTTON(sName := 'Voter 3' , sIconName := '', nThisTab := E_HMI_VOTER_TABS.VOTER_3);
    fbVoter4Button  : FB_HMI_BUTTON(sName := 'Voter 4' , sIconName := '', nThisTab := E_HMI_VOTER_TABS.VOTER_4);
    fbVoter5Button  : FB_HMI_BUTTON(sName := 'Voter 5' , sIconName := '', nThisTab := E_HMI_VOTER_TABS.VOTER_5);
    fbVoter6Button  : FB_HMI_BUTTON(sName := 'Voter 6' , sIconName := '', nThisTab := E_HMI_VOTER_TABS.VOTER_6);
    fbVoter7Button  : FB_HMI_BUTTON(sName := 'Voter 7' , sIconName := '', nThisTab := E_HMI_VOTER_TABS.VOTER_7);
    fbVoter8Button  : FB_HMI_BUTTON(sName := 'Voter 8' , sIconName := '', nThisTab := E_HMI_VOTER_TABS.VOTER_8);
    fbVoter9Button  : FB_HMI_BUTTON(sName := 'Voter 9' , sIconName := '', nThisTab := E_HMI_VOTER_TABS.VOTER_9);
    fbVoter10Button : FB_HMI_BUTTON(sName := 'Voter 10', sIconName := '', nThisTab := E_HMI_VOTER_TABS.VOTER_10);
    
    fbVoter1 : FB_HMI_VOTER;
    fbVoter2 : FB_HMI_VOTER;
    fbVoter3 : FB_HMI_VOTER;
    fbVoter4 : FB_HMI_VOTER;
    fbVoter5 : FB_HMI_VOTER;
    fbVoter6 : FB_HMI_VOTER;
    fbVoter7 : FB_HMI_VOTER;
    fbVoter8 : FB_HMI_VOTER;
    fbVoter9 : FB_HMI_VOTER;
    fbVoter10 : FB_HMI_VOTER;
END_VAR

fbHealthStatus(
    bIsEnabled := bConnected AND (
                   fbVoter1.fbHealthStatus.bEnabled
                OR fbVoter2.fbHealthStatus.bEnabled
                OR fbVoter3.fbHealthStatus.bEnabled
                OR fbVoter4.fbHealthStatus.bEnabled
                OR fbVoter5.fbHealthStatus.bEnabled
                OR fbVoter6.fbHealthStatus.bEnabled
                OR fbVoter7.fbHealthStatus.bEnabled
                OR fbVoter8.fbHealthStatus.bEnabled
                OR fbVoter9.fbHealthStatus.bEnabled
                OR fbVoter10.fbHealthStatus.bEnabled),
    bIsGood :=  (fbVoter1.fbHealthStatus.bGood OR NOT fbVoter1.fbHealthStatus.bEnabled)
            AND (fbVoter2.fbHealthStatus.bGood OR NOT fbVoter2.fbHealthStatus.bEnabled)
            AND (fbVoter3.fbHealthStatus.bGood OR NOT fbVoter3.fbHealthStatus.bEnabled)
            AND (fbVoter4.fbHealthStatus.bGood OR NOT fbVoter4.fbHealthStatus.bEnabled)
            AND (fbVoter5.fbHealthStatus.bGood OR NOT fbVoter5.fbHealthStatus.bEnabled)
            AND (fbVoter6.fbHealthStatus.bGood OR NOT fbVoter6.fbHealthStatus.bEnabled)
            AND (fbVoter7.fbHealthStatus.bGood OR NOT fbVoter7.fbHealthStatus.bEnabled)
            AND (fbVoter8.fbHealthStatus.bGood OR NOT fbVoter8.fbHealthStatus.bEnabled)
            AND (fbVoter9.fbHealthStatus.bGood OR NOT fbVoter9.fbHealthStatus.bEnabled)
            AND (fbVoter10.fbHealthStatus.bGood OR NOT fbVoter10.fbHealthStatus.bEnabled));

fbBusyStatus(
    bIsEnabled := bConnected,
    bIsBusy := FALSE);

fbVoter1(fbInstance := fbInstance.vote_img_1);
fbVoter2(fbInstance := fbInstance.vote_img_2);
fbVoter3(fbInstance := fbInstance.vote_img_3);
fbVoter4(fbInstance := fbInstance.vote_img_4);
fbVoter5(fbInstance := fbInstance.vote_img_5);
fbVoter6(fbInstance := fbInstance.vote_img_6);
fbVoter7(fbInstance := fbInstance.vote_img_7);
fbVoter8(fbInstance := fbInstance.vote_img_8);
fbVoter9(fbInstance := fbInstance.vote_img_9);
fbVoter10(fbInstance := fbInstance.vote_img_10);

